// TwinCAT 3 PLC project TcForge
// Title: TcForge
// Company: Home
// ProjectVersion: 2.0.0.0
// ProgramVersion: 3.1.4026.26
// libraries:
//   Tc2_Standard, 3.4.7.0 (Beckhoff Automation GmbH)
//   Tc2_System, 3.10.2.0 (Beckhoff Automation GmbH)
//   Tc3_Module, 3.4.7.0 (Beckhoff Automation GmbH)
// project tree:
//   POUs/Control/BangBang/ ST_BangBang_Cfg.TcDUT, FB_BangBang.TcPOU
//   POUs/Control/PID/ E_ControlReason.TcDUT, ST_PID_Full_Cfg.TcDUT, ST_PID_Full_Sts.TcDUT, FB_PID_Full.TcPOU
//   POUs/Control/Temperature/ ST_TempController_Cfg.TcDUT, ST_TempController_Sts.TcDUT, FB_TempController.TcPOU
//   POUs/Control/SwitchingPV/ E_PvSource.TcDUT, ST_SwitchingPvPid_Cfg.TcDUT, ST_SwitchingPvPid_Sts.TcDUT, FB_SwitchingPvPid.TcPOU
//   POUs/Control/Hysteresis/ E_HysteresisReason.TcDUT, ST_Hysteresis_Cfg.TcDUT, ST_Hysteresis_Sts.TcDUT, FB_HysteresisControl.TcPOU
//   POUs/Utilities/ FB_ExecutionContinuity.TcPOU, F_IsFiniteReal.TcPOU, F_IsFiniteLReal.TcPOU, F_GetTaskCycleTime.TcPOU, F_Now.TcPOU (not stored), FB_BitMatrix64.TcPOU, FB_LPF_FirstOrder_IIR.TcPOU
//   POUs/IO/Common/ E_IOHealthReason.TcDUT, FB_IOQualityMonitor.TcPOU (not stored), F_EtherCATSlaveDataValid.TcPOU, E_IO_Quality.TcDUT, E_Unit.TcDUT, U_IoRaw_In.TcDUT, U_IoRaw_Out.TcDUT (not stored)
//   POUs/Base/ FB_OperatorMailbox.TcPOU, ST_OperatorCommandRecord.TcDUT (not stored), E_OperatorCommand.TcDUT, E_Requester.TcDUT (not stored), E_RpcMethodResponse.TcDUT (not stored), F_ValidateRequester.TcPOU (not stored), FB_DeviceBase.TcPOU, ST_DeviceHeader_Sts.TcDUT (not stored), ST_FaultEntry.TcDUT (not stored)
//   POUs/Devices/Pneumatics/TwoPosActuator/ E_TwoPosActuator_Fault.TcDUT (not stored), E_TwoPosActuator_State.TcDUT (not stored), FB_TwoPosActuator.TcPOU, ST_TwoPosActuator_Cfg.TcDUT (not stored), ST_TwoPosActuator_Sts.TcDUT (not stored)
//   POUs/Logic/Interlocks/ FB_Interlock.TcPOU, ST_Interlock_Config.TcDUT, ST_Interlock_Status.TcDUT, ST_Interlock_Faceplate.TcDUT
//   POUs/Logic/Sequencing/Permissives/ FB_Permissives.TcPOU, ST_Permissive_Config.TcDUT (not stored), ST_Permissive_Status.TcDUT, ST_Permissive_Faceplate.TcDUT
//   POUs/Logic/Sequencing/StateMachine/ E_SM_Fault.TcDUT, E_SM_State.TcDUT, FB_StateMachine.TcPOU, FB_Step.TcPOU, ST_SM_Status.TcDUT, ST_SM_Step.TcDUT (not stored)
//   POUs/IO/DigitalInput/ FB_DigitalInput.TcPOU, ST_DigitalInput_Cfg.TcDUT, ST_DigitalInput_Sts.TcDUT, E_DigitalInput_Fault.TcDUT (not stored)
//   POUs/IO/DigitalOutput/ FB_DigitalOutput.TcPOU, ST_DigitalOutput_Cfg.TcDUT (not stored), ST_DigitalOutput_Sts.TcDUT, E_DigitalOutput_Fault.TcDUT, E_DigitalOutput_Mode.TcDUT
//   POUs/IO/AnalogInput/ FB_AnalogInput.TcPOU, ST_AnalogInput_Cfg.TcDUT, ST_AnalogInput_Sts.TcDUT, E_AnalogInput_Fault.TcDUT (not stored)
//   POUs/IO/AnalogOutput/ FB_AnalogOutput.TcPOU, ST_AnalogOutput_Cfg.TcDUT, ST_AnalogOutput_Sts.TcDUT, E_AnalogOutput_Fault.TcDUT (not stored)
//   POUs/Alarms/Common/ I_Alarm.TcIO (not stored), E_AlarmEvaluation.TcDUT (not stored), E_AlarmSeverity.TcDUT, ST_Alarm_Cfg.TcDUT (not stored), ST_Alarm_Sts.TcDUT, FB_AlarmBase.TcPOU
//   POUs/Alarms/Simple/ ST_AlarmSimple_Cfg.TcDUT, FB_AlarmSimple.TcPOU
//   POUs/Alarms/Threshold/ ST_AlarmThreshold_Cfg.TcDUT, FB_AlarmThreshold.TcPOU
//   POUs/Alarms/Limit/ ST_AlarmLimit_Cfg.TcDUT, ST_AlarmLimit_Sts.TcDUT, FB_AlarmLimit.TcPOU
//   POUs/Alarms/Deviation/ ST_AlarmDeviation_Cfg.TcDUT, FB_AlarmDeviation.TcPOU (not stored)
//   POUs/Alarms/RateOfChange/ ST_AlarmRateOfChange_Cfg.TcDUT, FB_AlarmRateOfChange.TcPOU
// real-time tasks:
//   TASK PlcTask: cycle T#10ms, priority 1, ADS port 350

// ---- POUs/Control/BangBang/ST_BangBang_Cfg.TcDUT
// The two CV values map a Boolean demand into engineering output units.
TYPE ST_BangBang_Cfg :
STRUCT
    hysteresis : ST_Hysteresis_Cfg;
    lowValue   : REAL := 0.0;
    highValue  : REAL := 100.0;
END_STRUCT
END_TYPE

// ---- POUs/Control/PID/E_ControlReason.TcDUT
// Controller state; an output device applies the physical safe level.
{attribute 'qualified_only'}
{attribute 'strict'}
TYPE E_ControlReason :
(
    Disabled      := 0,
    Automatic     := 1,
    Manual        := 2,
    Held          := 3,
    Tracking      := 4,
    BadQuality    := 5,
    InvalidValue  := 6,
    InvalidConfig := 7,
    InvalidTiming := 8,
    ConfigChanged := 9
);
END_TYPE

// ---- POUs/Control/PID/ST_PID_Full_Cfg.TcDUT
// All rates are engineering units per second. CV and integral limits are
// output units. A zero rate disables that directional ramp.
TYPE ST_PID_Full_Cfg :
STRUCT
    kp              : REAL := 1.0;
    ki              : REAL := 0.0; // Ideal form, 1/s.
    kd              : REAL := 0.0; // Ideal form, s.
    standardForm    : BOOL := FALSE;
    integralTime    : TIME := T#0MS; // Standard form; zero disables I.
    derivativeTime  : TIME := T#0MS; // Standard form; zero disables D.
    derivativeTau   : TIME := T#0MS; // Zero disables derivative filtering.
    reverseActing   : BOOL := FALSE;

    spMin           : REAL := -1E30;
    spMax           : REAL := 1E30;
    spRateUp        : REAL := 0.0;
    spRateDown      : REAL := 0.0;

    cvMin           : REAL := 0.0;
    cvMax           : REAL := 100.0;
    cvRateUp        : REAL := 0.0;
    cvRateDown      : REAL := 0.0;
    integralMin     : REAL := -100.0;
    integralMax     : REAL := 100.0;
    safeCv          : REAL := 0.0;

    cycleTime       : TIME := T#0MS; // Zero reads the owning task period.
    maxDt           : TIME := T#1S;  // Maximum declared task interval; not a missed-cycle detector.
END_STRUCT
END_TYPE

// ---- POUs/Control/PID/ST_PID_Full_Sts.TcDUT
// Calculation diagnostics. ready is FALSE when outCv carries safeCv.
TYPE ST_PID_Full_Sts :
STRUCT
    ready        : BOOL;
    reason       : E_ControlReason := E_ControlReason.Disabled;
    saturated    : BOOL;
    spRamping    : BOOL;
    cvRamping    : BOOL;
    spRequested  : REAL;
    spApplied    : REAL;
    pv           : REAL;
    cv           : REAL;
    error        : LREAL;
    pTerm        : LREAL;
    iTerm        : LREAL;
    dTerm        : LREAL;
END_STRUCT
END_TYPE

// ---- POUs/Control/Temperature/ST_TempController_Cfg.TcDUT
// Time-proportioning output for a heater, fan or SSR. Configure pid CV as
// 0..100 percent with safeCv=0; the wrapper rejects other CV ranges.
TYPE ST_TempController_Cfg :
STRUCT
    pid                 : ST_PID_Full_Cfg;
    pwmPeriod           : TIME := T#2S;
    standbyEnabled      : BOOL := FALSE;
    standbySetpoint     : REAL := 25.0;
END_STRUCT
END_TYPE

// ---- POUs/Control/Temperature/ST_TempController_Sts.TcDUT
TYPE ST_TempController_Sts :
STRUCT
    ready          : BOOL;
    standbyActive  : BOOL;
    dutyPercent    : REAL;
    pwmOn          : BOOL;
    pid            : ST_PID_Full_Sts;
END_STRUCT
END_TYPE

// ---- POUs/Control/SwitchingPV/E_PvSource.TcDUT
{attribute 'qualified_only'}
{attribute 'strict'}
TYPE E_PvSource :
(
    PV1 := 0,
    PV2 := 1
);
END_TYPE

// ---- POUs/Control/SwitchingPV/ST_SwitchingPvPid_Cfg.TcDUT
// Each sensor can have separate tuning and SP limits. Both configurations
// must have identical CV limits and safe CV because they drive one device.
TYPE ST_SwitchingPvPid_Cfg :
STRUCT
    pv1 : ST_PID_Full_Cfg;
    pv2 : ST_PID_Full_Cfg;
END_STRUCT
END_TYPE

// ---- POUs/Control/SwitchingPV/ST_SwitchingPvPid_Sts.TcDUT
TYPE ST_SwitchingPvPid_Sts :
STRUCT
    ready             : BOOL;
    activeSource      : E_PvSource := E_PvSource.PV1;
    sourceChanged     : BOOL;
    activePv          : REAL;
    cv                : REAL;
    pid               : ST_PID_Full_Sts;
END_STRUCT
END_TYPE

// ---- POUs/Control/Hysteresis/E_HysteresisReason.TcDUT
// Why a hysteresis controller is or is not evaluating a live measurement.
{attribute 'qualified_only'}
{attribute 'strict'}
TYPE E_HysteresisReason :
(
    Disabled      := 0,
    Ready         := 1,
    BadQuality    := 2,
    InvalidValue  := 3,
    InvalidConfig := 4
);
END_TYPE

// ---- POUs/Control/Hysteresis/ST_Hysteresis_Cfg.TcDUT
// Both thresholds use the same engineering unit as the conditioned PV.
// The default equal thresholds are deliberately invalid until configured.
TYPE ST_Hysteresis_Cfg :
STRUCT
    low        : REAL := 0.0;
    high       : REAL := 0.0;
    onBelowLow : BOOL := TRUE; // TRUE for heating/fill, FALSE for cooling/vent.
END_STRUCT
END_TYPE

// ---- POUs/Control/Hysteresis/ST_Hysteresis_Sts.TcDUT
// Diagnostic status only. The application connects outDemand to an owned
// output device and remains responsible for its interlocks and safe level.
TYPE ST_Hysteresis_Sts :
STRUCT
    ready      : BOOL;
    demand     : BOOL;
    inDeadband : BOOL;
    reason     : E_HysteresisReason := E_HysteresisReason.Disabled;
END_STRUCT
END_TYPE

// ---- POUs/IO/Common/E_IOHealthReason.TcDUT
{attribute 'qualified_only'}
{attribute 'strict'}
TYPE E_IOHealthReason : (Disabled := 0, NoSample := 1, Communication := 2, Device := 3,
    InvalidSample := 4, Stale := 5, InvalidConfig := 6, SequenceReset := 7, Good := 8) USINT;
END_TYPE

// ---- POUs/Base/E_OperatorCommand.TcDUT
{attribute 'qualified_only'}
{attribute 'strict'}
TYPE E_OperatorCommand : (Reset, Ack, SetValue, ForceSafe, SetOn, SetOff, Advance, Retract, Abort, Home, Pause, Proceed, Retry, Start, Stop); END_TYPE

// ---- POUs/Logic/Interlocks/ST_Interlock_Config.TcDUT
(*
Interlock Configuration Structure
=================================
Configuration for FB_Interlock. Latching is the defining behavior of an
interlock, so every mapped bit latches by default (no nLatch mask). Bits
can optionally be made bypassable via nBypassable.
*)
{attribute 'OPC.UA.DA' := '1'}
{attribute 'OPC.UA.DA.Access' := '1'}
{attribute 'OPC.UA.DA.StructuredType' := '1'}
TYPE ST_Interlock_Config :
STRUCT
    // Required bits cannot disappear when their producer stops running.
    nRequired : ULINT := 0;
	{attribute 'OPC.UA.DA.Description' := 'Bypass configuration bitmask (1=bypassable, 0=not bypassable)'}
	nBypassable : ULINT := 0;
	{attribute 'OPC.UA.DA.Description' := 'Human readable names for each interlock bit'}
	aNames : ARRAY[0..63] OF STRING(50);
END_STRUCT
END_TYPE

// ---- POUs/Logic/Interlocks/ST_Interlock_Status.TcDUT
(*
Interlock Status Structure
==========================
Status outputs for FB_Interlock.
*)
{attribute 'OPC.UA.DA' := '1'}
{attribute 'OPC.UA.DA.Access' := '1'}
{attribute 'OPC.UA.DA.StructuredType' := '1'}
TYPE ST_Interlock_Status :
STRUCT
    nMissing : ULINT; // Required but not refreshed within the mapping timeout.
	{attribute 'OPC.UA.DA.Description' := 'Overall status - TRUE when all interlocks are good'}
	bOK : BOOL := FALSE;
	{attribute 'OPC.UA.DA.Description' := 'Effective interlock status after latch + bypass (1=good, 0=bad)'}
	nInterlocks : ULINT := 0;
	{attribute 'OPC.UA.DA.Description' := 'Latched status - stays bad until Reset() (1=good, 0=latched bad)'}
	nLatched : ULINT := 0;
	{attribute 'OPC.UA.DA.Description' := 'Current bypass mask (1=bypassed, 0=not bypassed)'}
	nBypassMask : ULINT := 0;
	{attribute 'OPC.UA.DA.Description' := 'Bit index (0-63) of the first bit to trip, 999=no trips'}
	nFirstFailureBitIndex : UDINT := 999;
	{attribute 'OPC.UA.DA.Description' := 'Individual interlock faceplate data for HMI'}
	aFaceplates : ARRAY[0..63] OF ST_Interlock_Faceplate;
END_STRUCT
END_TYPE

// ---- POUs/Logic/Interlocks/ST_Interlock_Faceplate.TcDUT
(*
Interlock Faceplate Structure
=============================
Per-bit HMI data for a single interlock condition.
*)
{attribute 'OPC.UA.DA' := '1'}
{attribute 'OPC.UA.DA.Access' := '1'}
{attribute 'OPC.UA.DA.StructuredType' := '1'}
TYPE ST_Interlock_Faceplate :
STRUCT
	{attribute 'OPC.UA.DA.Description' := 'Human readable name of the interlock'}
	name : STRING(50);
	{attribute 'OPC.UA.DA.Description' := 'Effective status after latch + bypass (TRUE=good, FALSE=bad)'}
	ok : BOOL;
	{attribute 'OPC.UA.DA.Description' := 'Raw real-time condition (TRUE=good, FALSE=bad)'}
	live : BOOL;
	{attribute 'OPC.UA.DA.Description' := 'TRUE if currently latched bad (needs Reset)'}
	latched : BOOL;
	{attribute 'OPC.UA.DA.Description' := 'TRUE if this bit is actively mapped via MapInput'}
	mapped : BOOL;
	{attribute 'OPC.UA.DA.Description' := 'TRUE if this bit is currently bypassed'}
	bypassed : BOOL;
	{attribute 'OPC.UA.DA.Description' := 'TRUE if this bit is configured as bypassable'}
	bypassable : BOOL;
END_STRUCT
END_TYPE

// ---- POUs/Logic/Sequencing/Permissives/ST_Permissive_Status.TcDUT
(*
Permissive Status Structure
===========================
Contains all status outputs from permissive function block
*)
{attribute 'OPC.UA.DA' := '1'}
{attribute 'OPC.UA.DA.Access' := '1'}
{attribute 'OPC.UA.DA.StructuredType' := '1'}
TYPE ST_Permissive_Status :
STRUCT
    nMissing : ULINT; // Required but not refreshed within the mapping timeout.
	{attribute 'OPC.UA.DA.Description' := 'Overall status - TRUE when all permissive bits are good'}
	bOK : BOOL := FALSE;
	{attribute 'OPC.UA.DA.Description' := 'Current permissive status after logic (1=good, 0=bad)'}
	nPermissives : ULINT := 0;
	{attribute 'OPC.UA.DA.Description' := 'Current bypass mask (1=bypassed, 0=not bypassed)'}
	nBypassMask : ULINT := 0;
	{attribute 'OPC.UA.DA.Description' := 'Bit index (0-63) of the first failure, 999=no failures'}
	nFirstFailureBitIndex : UDINT := 999;
	
	{attribute 'OPC.UA.DA.Description' := 'Individual permissive faceplate data for HMI'}
	aFaceplates : ARRAY[0..63] OF ST_Permissive_Faceplate;
END_STRUCT
END_TYPE

// ---- POUs/Logic/Sequencing/Permissives/ST_Permissive_Faceplate.TcDUT
(*
Permissive Faceplate Structure
==============================
Individual permissive bit information for HMI faceplate display
*)
{attribute 'OPC.UA.DA' := '1'}
{attribute 'OPC.UA.DA.Access' := '1'}
{attribute 'OPC.UA.DA.StructuredType' := '1'}
TYPE ST_Permissive_Faceplate :
STRUCT
	{attribute 'OPC.UA.DA.Description' := 'Human readable name of the permissive'}
	name : STRING(50);
	{attribute 'OPC.UA.DA.Description' := 'Real-time status of this permissive bit (TRUE=good, FALSE=bad)'}
	ok : BOOL;
	{attribute 'OPC.UA.DA.Description' := 'TRUE if this bit is actively mapped via MapInput'}
	mapped : BOOL;
	{attribute 'OPC.UA.DA.Description' := 'TRUE if this bit is currently bypassed'}
	bypassed : BOOL;
	{attribute 'OPC.UA.DA.Description' := 'TRUE if this bit is configured as bypassable'}
	bypassable : BOOL;
END_STRUCT
END_TYPE

// ---- POUs/Logic/Sequencing/StateMachine/E_SM_Fault.TcDUT
{attribute 'qualified_only'}
{attribute 'to_string'}
// Fault codes surfaced by FB_StateMachine through ST_DeviceHeader_Sts (the
// fault book-keeping lives on FB_DeviceBase). Range convention mirrors
// E_RpcMethodResponse so codes are self-documenting:
//
//   0        No fault
//   1-9      Timeouts
//   10-19    Feedback / hardware
//   20-29    State violations
//   30-39    Configuration
//   50-59    Interlocks / permissives
//   70-79    Submodule / propagation
//   100+     Device / application custom
//
// HMI displays ResolveFaultString(code) for the stable title and faultReason
// for the contextual detail (step number, step name, free-form operator
// message). Both live in ST_DeviceHeader_Sts.
TYPE E_SM_Fault :
(
    None                    := 0,

    StepTimeout             := 1,    // FB_Step.tonTimeout expired
    OddStepReached          := 2,    // default fault when a step moves onto an odd step number
    StepUserFault           := 3,    // user called step.RaiseFault(code, reason)

    InvalidStepConfiguration := 30,
    MissingStepImplementation := 31,
    DuplicateStepImplementation := 32,
    ShutdownFailed := 33,

    RunningInterlockTripped := 50,   // intlkRunning tripped, auto-aborted

    SubmoduleFaulted        := 70    // external inpSubmoduleFaulted asserted
);
END_TYPE

// ---- POUs/Logic/Sequencing/StateMachine/E_SM_State.TcDUT
{attribute 'qualified_only'}
{attribute 'strict'}
{attribute 'to_string'}
// Minimum useful set of machine states.
//
// Waiting states (quiescent, no sequence driving outputs):
//     STOPPED  - power-on default, not homed. Entry from Abort is STOPPED with Status.Faulted = TRUE.
//     READY    - homed and either just-homed or just-completed a cycle. LastState distinguishes the two.
//     PAUSED   - frozen mid-cycle, context held for Proceed.
//
// Active states (a step sequence is executing):
//     HOMING      (steps 1000-1999)
//     RUNNING     (steps 3000-3999)
//     STOPPING    (steps 2000-2999) - graceful shutdown sequence
//     ABORTING    (steps 5000-5999) - fast-safe shutdown sequence
//     PAUSING     (steps 4000-4999) - park motion / save context
//     PROCEEDING  (steps 6000-6999) - restore context / resume
TYPE E_SM_State :
(
    STOPPED     := 0,
    RUNNING     := 1,
    STOPPING    := 2,
    HOMING      := 4,
    ABORTING    := 8,
    READY       := 16,
    PAUSING     := 32,
    PAUSED      := 64,
    PROCEEDING  := 128
);
END_TYPE

// ---- POUs/Logic/Sequencing/StateMachine/ST_SM_Status.TcDUT
(*
Aggregated status published by FB_StateMachine. Contains the common device
header, the current state, derived readiness flags, OEE condition codes,
and the active step snapshot (ST_SM_Step).
*)
{attribute 'OPC.UA.DA' := '1'}
{attribute 'OPC.UA.DA.Access' := '1'}
{attribute 'OPC.UA.DA.StructuredType' := '1'}
TYPE ST_SM_Status :
STRUCT
    // Common device header (ready/busy/faulted, fault codes + strings, timestamps).
    header : ST_DeviceHeader_Sts;

    // Current state (enum with to_string for HMI)
    State : E_SM_State := E_SM_State.STOPPED;
    LastState : E_SM_State := E_SM_State.STOPPED;

    // Derived state categories
    ActiveState : BOOL;
    WaitingState : BOOL;

    // Computed fault flags
    Faulted : BOOL; // Always the base device fault state.
    AtRecoveryStep : BOOL; // Odd-numbered recovery step, independent of fault storage.
    SubmoduleFaulted : BOOL;
    ShutdownFailed : BOOL; // Abort failed; STOPPED does not imply confirmed physical shutdown.
    FailedStep : DINT; // Last failed step, cleared only by a successful Reset.

    // Permission-derived readiness
    ReadyToHome : BOOL;
    ReadyToStart : BOOL;
    ReadyToProceed : BOOL;

    // Auto-run tracking
    AutoCycleRequest : BOOL;

    // OEE condition codes (0 = clear, non-zero = active reason code)
    BlockedCondition : DINT;
    StarvedCondition : DINT;

    // Active step snapshot
    Step : ST_SM_Step;
END_STRUCT
END_TYPE

// ---- POUs/IO/DigitalInput/ST_DigitalInput_Cfg.TcDUT
// Configuration for FB_DigitalInput. All fields are configurable; defaults
// yield a plain pass-through of the physical signal.
{attribute 'OPC.UA.DA' := '1'}
{attribute 'OPC.UA.DA.Access' := '1'}
{attribute 'OPC.UA.DA.StructuredType' := '1'}
TYPE ST_DigitalInput_Cfg :
STRUCT
    // Signal conditioning
    {attribute 'OPC.UA.DA.Description' := 'Invert input signal (active-low sensors)'}
    invert            : BOOL := FALSE;

    // Asymmetric debounce: separate delays for each edge so a noisy 24 V
    // signal can have e.g. a 20 ms ON-delay but 0 ms OFF-delay. Set both to
    // T#0MS to disable.
    {attribute 'OPC.UA.DA.Description' := 'Rising-edge debounce delay (ON)'}
    debounceOn        : TIME := T#0MS;
    {attribute 'OPC.UA.DA.Description' := 'Falling-edge debounce delay (OFF)'}
    debounceOff       : TIME := T#0MS;

    // Quality watchdog: if inpQuality stays BAD for this long the FB raises
    // E_DigitalInput_Fault.BadQuality. T#0MS disables the watchdog.
    {attribute 'OPC.UA.DA.Description' := 'Raise BadQuality fault after this long in BAD quality (T#0MS = disabled)'}
    qualityFaultAfter : TIME := T#0MS;
END_STRUCT
END_TYPE

// ---- POUs/IO/DigitalInput/ST_DigitalInput_Sts.TcDUT
// Status of FB_DigitalInput. `header` is shared with every other device FB
// (see ST_DeviceHeader_Sts); device-specific fields sit below.
{attribute 'OPC.UA.DA' := '1'}
{attribute 'OPC.UA.DA.Access' := '1'}
{attribute 'OPC.UA.DA.StructuredType' := '1'}
TYPE ST_DigitalInput_Sts :
STRUCT
    header        : ST_DeviceHeader_Sts;

    {attribute 'OPC.UA.DA.Description' := 'Final processed value (after invert + debounce)'}
    value      : BOOL;
    {attribute 'OPC.UA.DA.Description' := 'Raw terminal reading (before invert / debounce)'}
    rawValue   : BOOL;
    {attribute 'OPC.UA.DA.Description' := 'Signal quality tag'}
    quality    : E_IO_Quality := E_IO_Quality.UNKNOWN;
    {attribute 'OPC.UA.DA.Description' := 'One-scan pulse on debounced rising edge'}
    risingEdge : BOOL;
    {attribute 'OPC.UA.DA.Description' := 'One-scan pulse on debounced falling edge'}
    fallingEdge: BOOL;
END_STRUCT
END_TYPE

// ---- POUs/IO/DigitalOutput/ST_DigitalOutput_Sts.TcDUT
// Status of FB_DigitalOutput. `header` is shared with every other device FB
// (see ST_DeviceHeader_Sts); device-specific fields sit below.
{attribute 'OPC.UA.DA' := '1'}
{attribute 'OPC.UA.DA.Access' := '1'}
{attribute 'OPC.UA.DA.StructuredType' := '1'}
TYPE ST_DigitalOutput_Sts :
STRUCT
    outputInhibited : BOOL;
    header        : ST_DeviceHeader_Sts;

    {attribute 'OPC.UA.DA.Description' := 'Final physical output value (after mode + invert)'}
    value      : BOOL;
    {attribute 'OPC.UA.DA.Description' := 'Last commanded value (survives power cycle)'}
    commanded  : BOOL;
    {attribute 'OPC.UA.DA.Description' := 'Signal quality tag'}
    quality    : E_IO_Quality := E_IO_Quality.UNKNOWN;
    {attribute 'OPC.UA.DA.Description' := 'One-scan pulse on physical output rising edge'}
    risingEdge : BOOL;
    {attribute 'OPC.UA.DA.Description' := 'One-scan pulse on physical output falling edge'}
    fallingEdge: BOOL;
END_STRUCT
END_TYPE

// ---- POUs/IO/AnalogInput/ST_AnalogInput_Cfg.TcDUT
// Configuration for FB_AnalogInput. Defaults provide numeric 0..100 scaling of
// an INT terminal scaled linearly from raw 0..32767 — adjust for the real
// hardware.
//
// FB_AnalogInput is intentionally conditioning-only: raw type select, quality
// gate, clamp-to-scaling-range, linear scale, optional LPF. If you need HH /
// HI / LO / LL process alarms, compose FB_AlarmLimit with the published
// value — that keeps alarm config, latching, severity, and ack logic in
// one place (see docs/8-Alarms.md).
{attribute 'OPC.UA.DA' := '1'}
{attribute 'OPC.UA.DA.Access' := '1'}
{attribute 'OPC.UA.DA.StructuredType' := '1'}
TYPE ST_AnalogInput_Cfg :
STRUCT
    // Which UNION member to read. Supported values:
    //   TYPE_REAL, TYPE_INT, TYPE_UINT, TYPE_WORD, TYPE_DWORD, TYPE_UDINT, TYPE_DINT
    {attribute 'OPC.UA.DA.Description' := 'Terminal numeric type (selects UNION member)'}
    inputType          : __SYSTEM.TYPE_CLASS := __SYSTEM.TYPE_CLASS.TYPE_INT;

    // When TRUE, the FB skips clamping + scaling + filtering and publishes
    // the raw REAL representation directly. Handy for soft signals, bit-
    // masked terminals, or diagnostics.
    {attribute 'OPC.UA.DA.Description' := 'Bypass clamp + scale + filter; publish raw value'}
    useRawValue        : BOOL := FALSE;

    // Raw-to-EU linear scaling. Example: 4-20 mA on an EL3024 reports raw
    // in [0, 32767]; to get 0-100 % set fRawMin=0, fRawMax=32767, fPvMin=0,
    // fPvMax=100.
    {attribute 'OPC.UA.DA.Description' := 'Raw value corresponding to fPvMin'}
    rawMin             : REAL := 0.0;
    {attribute 'OPC.UA.DA.Description' := 'Raw value corresponding to fPvMax'}
    rawMax             : REAL := 32767.0;

    {attribute 'OPC.UA.DA.Description' := 'Engineering value at fRawMin'}
    euMin              : REAL := 0.0;
    {attribute 'OPC.UA.DA.Description' := 'Engineering value at fRawMax'}
    euMax              : REAL := 100.0;
    {attribute 'OPC.UA.DA.Description' := 'Engineering-unit display metadata; configure explicitly'}
    unit               : E_Unit := E_Unit.UNSPECIFIED;

    // Clamp reporting. sts.clamped* always tracks whether the raw input
    // was outside [rawMin, rawMax]; clampAsFault promotes that condition
    // to a persistent device fault.
    {attribute 'OPC.UA.DA.Description' := 'Promote out-of-range raw readings to ClampLow / ClampHigh faults'}
    clampAsFault       : BOOL := FALSE;

    // Optional first-order low-pass filter. T#0MS disables filtering.
    {attribute 'OPC.UA.DA.Description' := 'Low-pass filter time constant (T#0MS = disabled)'}
    filterTau          : TIME := T#0MS;

    // Quality watchdog.
    {attribute 'OPC.UA.DA.Description' := 'Raise BadQuality fault after this long in BAD quality (T#0MS = disabled)'}
    qualityFaultAfter  : TIME := T#0MS;
END_STRUCT
END_TYPE

// ---- POUs/IO/AnalogInput/ST_AnalogInput_Sts.TcDUT
// Status of FB_AnalogInput. `header` is shared with every device FB;
// device-specific fields sit below. Process-alarm status (HH/HI/LO/LL) is
// not part of this surface — use FB_AlarmLimit composed with value.
{attribute 'OPC.UA.DA' := '1'}
{attribute 'OPC.UA.DA.Access' := '1'}
{attribute 'OPC.UA.DA.StructuredType' := '1'}
TYPE ST_AnalogInput_Sts :
STRUCT
    header          : ST_DeviceHeader_Sts;

    {attribute 'OPC.UA.DA.Description' := 'Final value in engineering units (after clamp, scale, filter)'}
    value        : REAL;
    {attribute 'OPC.UA.DA.Description' := 'Raw value as REAL, before clamping and scaling'}
    rawReal      : REAL;
    {attribute 'OPC.UA.DA.Description' := 'Scaled value (EU), before filter'}
    scaled       : REAL;
    {attribute 'OPC.UA.DA.Description' := 'Echo of cfg.unit for HMI consumption'}
    unit         : E_Unit := E_Unit.UNSPECIFIED;
    {attribute 'OPC.UA.DA.Description' := 'Signal quality tag (may be promoted to CLAMPED)'}
    quality      : E_IO_Quality := E_IO_Quality.UNKNOWN;

    {attribute 'OPC.UA.DA.Description' := 'Raw below configured RawMin'}
    clampedLow   : BOOL;
    {attribute 'OPC.UA.DA.Description' := 'Raw above configured RawMax'}
    clampedHigh  : BOOL;
    {attribute 'OPC.UA.DA.Description' := 'Either clamp direction active'}
    clampActive  : BOOL;
END_STRUCT
END_TYPE

// ---- POUs/IO/AnalogOutput/ST_AnalogOutput_Cfg.TcDUT
// Configuration for FB_AnalogOutput. Defaults drive a numeric 0..100 command
// range into an INT 0..32767 scaled terminal.
{attribute 'OPC.UA.DA' := '1'}
{attribute 'OPC.UA.DA.Access' := '1'}
{attribute 'OPC.UA.DA.StructuredType' := '1'}
TYPE ST_AnalogOutput_Cfg :
STRUCT
    // Startup restoration requires explicit application opt-in.
    restoreCommandOnRestart : BOOL := FALSE;
    // Optional hold during bad/unknown quality. Recovery still requires a fresh command.
    holdOnBadQuality : BOOL := FALSE;
    safeRaw : REAL := 0.0; // Terminal units, independent of scaling.
    // Which UNION member to write. Supported values:
    //   TYPE_REAL, TYPE_INT, TYPE_UINT, TYPE_WORD, TYPE_DWORD, TYPE_UDINT, TYPE_DINT
    {attribute 'OPC.UA.DA.Description' := 'Terminal numeric type (selects UNION member)'}
    outputType         : __SYSTEM.TYPE_CLASS := __SYSTEM.TYPE_CLASS.TYPE_INT;

    // When TRUE, the FB writes the command REAL directly into the UNION
    // without clamping or scaling. Handy for soft signals / diagnostics.
    {attribute 'OPC.UA.DA.Description' := 'Write commanded value directly; skip clamp + scale'}
    useRawValue        : BOOL := FALSE;

    // Command limits in engineering units.
    {attribute 'OPC.UA.DA.Description' := 'Minimum allowed command (EU)'}
    minCv              : REAL := 0.0;
    {attribute 'OPC.UA.DA.Description' := 'Maximum allowed command (EU)'}
    maxCv              : REAL := 100.0;

    // EU <-> raw linear scaling.
    {attribute 'OPC.UA.DA.Description' := 'Engineering value at fRawMin'}
    euMin              : REAL := 0.0;
    {attribute 'OPC.UA.DA.Description' := 'Engineering value at fRawMax'}
    euMax              : REAL := 100.0;
    {attribute 'OPC.UA.DA.Description' := 'Raw value at fEuMin'}
    rawMin             : REAL := 0.0;
    {attribute 'OPC.UA.DA.Description' := 'Raw value at fEuMax'}
    rawMax             : REAL := 32767.0;
    {attribute 'OPC.UA.DA.Description' := 'Engineering-unit display metadata; configure explicitly'}
    unit               : E_Unit := E_Unit.UNSPECIFIED;

    // Clamp alarm behaviour.
    {attribute 'OPC.UA.DA.Description' := 'Promote clamping to a device fault (ClampLow / ClampHigh)'}
    clampAsFault       : BOOL := FALSE;

    // Quality watchdog.
    {attribute 'OPC.UA.DA.Description' := 'Raise BadQuality fault after this long in BAD quality (T#0MS = disabled)'}
    qualityFaultAfter  : TIME := T#0MS;
END_STRUCT
END_TYPE

// ---- POUs/IO/AnalogOutput/ST_AnalogOutput_Sts.TcDUT
// Status of FB_AnalogOutput. `header` is shared with every device FB;
// device-specific fields sit below.
{attribute 'OPC.UA.DA' := '1'}
{attribute 'OPC.UA.DA.Access' := '1'}
{attribute 'OPC.UA.DA.StructuredType' := '1'}
TYPE ST_AnalogOutput_Sts :
STRUCT
    outputInhibited : BOOL; // value (EU) is not valid when inhibited; rawReal is the applied fallback/held raw value.
    header        : ST_DeviceHeader_Sts;

    {attribute 'OPC.UA.DA.Description' := 'Clamped command actually written (EU)'}
    value      : REAL;
    {attribute 'OPC.UA.DA.Description' := 'Last commanded value before clamping (EU, survives power cycle)'}
    commanded  : REAL;
    {attribute 'OPC.UA.DA.Description' := 'Raw value written to the terminal (REAL view of the UNION)'}
    rawReal    : REAL;
    {attribute 'OPC.UA.DA.Description' := 'Echo of cfg.unit for HMI consumption'}
    unit       : E_Unit := E_Unit.UNSPECIFIED;
    {attribute 'OPC.UA.DA.Description' := 'Signal quality tag'}
    quality    : E_IO_Quality := E_IO_Quality.UNKNOWN;

    {attribute 'OPC.UA.DA.Description' := 'Command clamped at MinCv'}
    clampedLow : BOOL;
    {attribute 'OPC.UA.DA.Description' := 'Command clamped at MaxCv'}
    clampedHigh: BOOL;
    {attribute 'OPC.UA.DA.Description' := 'Either clamp direction active'}
    clampActive: BOOL;
END_STRUCT
END_TYPE

// ---- POUs/IO/DigitalOutput/E_DigitalOutput_Fault.TcDUT
{attribute 'qualified_only'}
{attribute 'to_string'}
// Fault codes for FB_DigitalOutput. Range convention matches the shared
// device-fault convention (see docs/2-Architecture.md):
//   0        No fault
//   1-9      Timeouts
//   10-19    Feedback / hardware / signal
//   20-29    State violations
//   40-49    Configuration / process limits
//   50-59    Interlocks / permissives
TYPE E_DigitalOutput_Fault :
(
    None        := 0,

    BadConfig := 40,
    BadQuality  := 10     // outgoing signal not writable (quality latched BAD past cfg.tQualityFaultAfter)
);
END_TYPE

// ---- POUs/IO/DigitalOutput/E_DigitalOutput_Mode.TcDUT
// Output shaping modes for FB_DigitalOutput.
//   Regular         : output tracks the commanded value (optionally inverted)
//   SinglePulse     : one-shot — commanded rising edge drives the output ON
//                     for cfg.tPulseOn, then OFF
//   ContinuousPulse : while commanded TRUE, output cycles ON/OFF with
//                     cfg.tPulseOn / cfg.tPulseOff (good for lamps, blinkers,
//                     repeat-start pulses)
{attribute 'qualified_only'}
{attribute 'strict'}
{attribute 'to_string'}
TYPE E_DigitalOutput_Mode :
(
    Regular         := 0,
    SinglePulse     := 1,
    ContinuousPulse := 2
);
END_TYPE

// ---- POUs/IO/Common/E_IO_Quality.TcDUT
// Signal quality tag carried by every IO block's status. The value lets the
// HMI and downstream logic react to wire breaks, out-of-range readings, or
// sensor faults without each consumer reinventing its own "is this bit /
// reading trustworthy?" logic.
//
// Meaning:
//   UNKNOWN : block has not evaluated yet (first scan, or no data source)
//   BAD     : signal is not usable (wire break, TwinCAT WcState, etc.)
//   GOOD    : signal is valid and within configured range
//   CLAMPED : signal is valid but was forced to the scaling limit
//
// Some device inputs default to GOOD for software signals. Hardware applications
// must explicitly supply quality from diagnostics, e.g. FB_IOQualityMonitor.
{attribute 'qualified_only'}
{attribute 'strict'}
{attribute 'to_string'}
TYPE E_IO_Quality :
(
    UNKNOWN := 0,
    BAD     := 1,
    GOOD    := 2,
    CLAMPED := 3
) USINT;
END_TYPE

// ---- POUs/IO/Common/E_Unit.TcDUT
// Display metadata for analog IO. The value is already scaled by the owning
// device; this enum does not convert or validate engineering units. An HMI may
// map the enum to a symbol (for example MILLIMETER -> mm).
//
// Keep explicit numeric values stable after publication because OPC clients may
// store them. Extend for machine-relevant measurements; never repurpose a code.
{attribute 'qualified_only'}
{attribute 'strict'}
{attribute 'to_string'}
TYPE E_Unit :
(
    // A channel whose display unit has not been configured.
    UNSPECIFIED                   := 0,

    // Ratio and discrete quantity.
    PERCENT                       := 1,     // %
    COUNT                         := 2,     // pieces / cycles

    // Position, orientation, velocity and acceleration.
    MILLIMETER                    := 3,     // mm
    MICROMETER                    := 4,     // um
    DEGREE                        := 5,     // angular degrees
    MILLIMETER_PER_SECOND         := 6,     // mm/s
    MILLIMETER_PER_SECOND_SQUARED := 7,     // mm/s^2
    RPM                           := 8,     // revolutions/minute

    // Force, torque, mass and pneumatic pressure.
    NEWTON                        := 9,     // N
    NEWTON_METER                  := 10,    // N m
    GRAM                          := 11,    // g
    KILOGRAM                      := 12,    // kg
    BAR                           := 13,    // bar
    KILOPASCAL                    := 14,    // kPa

    // Temperature and electrical measurements.
    DEGREE_CELSIUS                := 15,    // deg C
    DEGREE_FAHRENHEIT             := 16,    // deg F
    VOLTS                         := 17,    // V
    AMPS                          := 18,    // A
    WATT                          := 19,    // W
    HERTZ                         := 20,    // Hz

    // Cycle measurements and sensor-reported durations.
    SECOND                        := 21,    // s
    MILLISECOND                   := 22     // ms
);
END_TYPE

// ---- POUs/IO/Common/U_IoRaw_In.TcDUT
// Raw terminal representation. The application owns hardware mapping.
TYPE U_IoRaw_In :
UNION
    dw    : DWORD;
    fReal : REAL;
    w     : WORD;
    nInt  : INT;
    ui    : UINT;
    di    : DINT;
    udi   : UDINT;
END_UNION
END_TYPE

// ---- POUs/Alarms/Common/E_AlarmSeverity.TcDUT
// HMI / stacklight severity tag carried by every alarm status.
// Numeric order is meaningful — aggregators MAX() across alarms to pick the
// highest tier that's currently active.
{attribute 'qualified_only'}
{attribute 'strict'}
{attribute 'to_string'}
TYPE E_AlarmSeverity :
(
    NONE     := 0,   // bookkeeping: alarm disabled or inactive
    INFO     := 1,   // informational, no operator action required
    WARNING  := 2,   // operator should investigate
    CRITICAL := 3,   // urgent; process may be about to lose control
    SHUTDOWN := 4    // interlock-grade; a controller is already acting
) USINT;
END_TYPE

// ---- POUs/Alarms/Common/ST_Alarm_Sts.TcDUT
// Uniform alarm status. Every FB_Alarm* fills this struct identically so
// HMIs and aggregators can bind to any alarm generically.
{attribute 'OPC.UA.DA' := '1'}
{attribute 'OPC.UA.DA.Access' := '1'}
{attribute 'OPC.UA.DA.StructuredType' := '1'}
TYPE ST_Alarm_Sts :
STRUCT
    // Valid fresh evaluation; active may remain held while validity is false.
    valid : BOOL;
    evaluationState : E_AlarmEvaluation := E_AlarmEvaluation.Disabled;
    {attribute 'OPC.UA.DA.Description' := 'Echo of cfg.bEnable'}
    enabled    : BOOL;

    {attribute 'OPC.UA.DA.Description' := 'Instantaneous condition before debounce'}
    raw        : BOOL;

    {attribute 'OPC.UA.DA.Description' := 'After tOnDelay / tOffDelay'}
    debounced  : BOOL;

    {attribute 'OPC.UA.DA.Description' := 'Public is-it-firing bit (latch when bRequireAck)'}
    active     : BOOL;

    {attribute 'OPC.UA.DA.Description' := 'TRUE while latch is awaiting Ack()'}
    latched    : BOOL;

    {attribute 'OPC.UA.DA.Description' := 'TRUE once the current latch has been acknowledged'}
    acked      : BOOL;

    {attribute 'OPC.UA.DA.Description' := 'Severity while active; NONE while inactive'}
    eSeverity     : E_AlarmSeverity := E_AlarmSeverity.NONE;

    {attribute 'OPC.UA.DA.Description' := 'Echo of cfg.sMessage'}
    sMessage      : STRING(79);

    {attribute 'OPC.UA.DA.Description' := 'Who acknowledged the current latch'}
    ackRequester  : E_Requester;

    {attribute 'OPC.UA.DA.Description' := 'Last rising edge of debounced (LTIME)'}
    tsTripped     : LTIME;

    {attribute 'OPC.UA.DA.Description' := 'Last falling edge of debounced (LTIME)'}
    tsCleared     : LTIME;

    {attribute 'OPC.UA.DA.Description' := 'Last accepted Ack() timestamp (LTIME)'}
    tsAcked       : LTIME;
END_STRUCT
END_TYPE

// ---- POUs/Alarms/Simple/ST_AlarmSimple_Cfg.TcDUT
// Config for FB_AlarmSimple — no extra knobs beyond the shared common head.
{attribute 'OPC.UA.DA' := '1'}
{attribute 'OPC.UA.DA.Access' := '1'}
{attribute 'OPC.UA.DA.StructuredType' := '1'}
TYPE ST_AlarmSimple_Cfg :
STRUCT
    {attribute 'OPC.UA.DA.Description' := 'Shared alarm configuration (enable, delays, ack, severity, message)'}
    common : ST_Alarm_Cfg;
END_STRUCT
END_TYPE

// ---- POUs/Alarms/Threshold/ST_AlarmThreshold_Cfg.TcDUT
// Config for FB_AlarmThreshold. Single-direction REAL threshold check.
// Rule: strict > / < (exact threshold value does not trip).
// Exactly one direction must be selected while enabled; otherwise InvalidConfig.
{attribute 'OPC.UA.DA' := '1'}
{attribute 'OPC.UA.DA.Access' := '1'}
{attribute 'OPC.UA.DA.StructuredType' := '1'}
TYPE ST_AlarmThreshold_Cfg :
STRUCT
    {attribute 'OPC.UA.DA.Description' := 'Shared alarm configuration'}
    common     : ST_Alarm_Cfg;

    {attribute 'OPC.UA.DA.Description' := 'Threshold value to compare inpValue against'}
    fThreshold : REAL := 0.0;

    {attribute 'OPC.UA.DA.Description' := 'TRUE = trip when inpValue > fThreshold'}
    bFailHigh  : BOOL := FALSE;

    {attribute 'OPC.UA.DA.Description' := 'TRUE = trip when inpValue < fThreshold'}
    bFailLow   : BOOL := FALSE;
END_STRUCT
END_TYPE

// ---- POUs/Alarms/Limit/ST_AlarmLimit_Cfg.TcDUT
// Four-level limit ladder: HiHi / Hi / Lo / LoLo. Each level is a full
// ST_AlarmThreshold_Cfg, so each can have its own delay, severity, ack
// requirement, and message. Remember every level defaults to bEnable := FALSE.
{attribute 'OPC.UA.DA' := '1'}
{attribute 'OPC.UA.DA.Access' := '1'}
{attribute 'OPC.UA.DA.StructuredType' := '1'}
TYPE ST_AlarmLimit_Cfg :
STRUCT
    {attribute 'OPC.UA.DA.Description' := 'High-High (critical high, e.g. emergency shutdown)'}
    HiHi : ST_AlarmThreshold_Cfg;

    {attribute 'OPC.UA.DA.Description' := 'High (warning high, operator alert)'}
    Hi   : ST_AlarmThreshold_Cfg;

    {attribute 'OPC.UA.DA.Description' := 'Low (warning low)'}
    Lo   : ST_AlarmThreshold_Cfg;

    {attribute 'OPC.UA.DA.Description' := 'Low-Low (critical low)'}
    LoLo : ST_AlarmThreshold_Cfg;
END_STRUCT
END_TYPE

// ---- POUs/Alarms/Limit/ST_AlarmLimit_Sts.TcDUT
// Status for FB_AlarmLimit. Each level has its own raw ST_Alarm_Sts so the
// HMI can show full forensics per tier. The top-level *Suppressed* flags apply
// flooding suppression: HiHi suppresses Hi, LoLo suppresses Lo — so the HMI
// can pick exactly one active level per direction.
{attribute 'OPC.UA.DA' := '1'}
{attribute 'OPC.UA.DA.Access' := '1'}
{attribute 'OPC.UA.DA.StructuredType' := '1'}
TYPE ST_AlarmLimit_Sts :
STRUCT
    // Valid fresh evaluation; active may remain held while validity is false.
    valid : BOOL;
    evaluationState : E_AlarmEvaluation := E_AlarmEvaluation.Disabled;
    {attribute 'OPC.UA.DA.Description' := 'HiHi sub-alarm status'}
    HiHi : ST_Alarm_Sts;
    {attribute 'OPC.UA.DA.Description' := 'Hi sub-alarm status'}
    Hi   : ST_Alarm_Sts;
    {attribute 'OPC.UA.DA.Description' := 'Lo sub-alarm status'}
    Lo   : ST_Alarm_Sts;
    {attribute 'OPC.UA.DA.Description' := 'LoLo sub-alarm status'}
    LoLo : ST_Alarm_Sts;

    {attribute 'OPC.UA.DA.Description' := 'HiHi active (rollup after suppression)'}
    hiHiActive : BOOL;
    {attribute 'OPC.UA.DA.Description' := 'Hi active and not suppressed by HiHi'}
    hiActive   : BOOL;
    {attribute 'OPC.UA.DA.Description' := 'Lo active and not suppressed by LoLo'}
    loActive   : BOOL;
    {attribute 'OPC.UA.DA.Description' := 'LoLo active (rollup after suppression)'}
    loLoActive : BOOL;

    {attribute 'OPC.UA.DA.Description' := 'Any of the four levels currently active'}
    anyActive  : BOOL;
    {attribute 'OPC.UA.DA.Description' := 'Highest severity across all active levels'}
    eSeverity     : E_AlarmSeverity;
END_STRUCT
END_TYPE

// ---- POUs/Alarms/Deviation/ST_AlarmDeviation_Cfg.TcDUT
// Config for FB_AlarmDeviation. Two modes, selected by bUseSetpoint.
//
//   Absolute (bUseSetpoint = FALSE, default):
//       trip = inpPv > fHighLimit OR inpPv < fLowLimit
//       inpSetpoint is ignored
//
//   Setpoint deviation (bUseSetpoint = TRUE):
//       trip = inpPv > (inpSetpoint + fHighLimit) OR inpPv < (inpSetpoint - fLowLimit)
//       High/Low limits are asymmetric deviations from setpoint.
{attribute 'OPC.UA.DA' := '1'}
{attribute 'OPC.UA.DA.Access' := '1'}
{attribute 'OPC.UA.DA.StructuredType' := '1'}
TYPE ST_AlarmDeviation_Cfg :
STRUCT
    {attribute 'OPC.UA.DA.Description' := 'Shared alarm configuration'}
    common       : ST_Alarm_Cfg;

    {attribute 'OPC.UA.DA.Description' := 'Absolute high limit, or +deviation when bUseSetpoint = TRUE'}
    fHighLimit   : REAL := 0.0;

    {attribute 'OPC.UA.DA.Description' := 'Absolute low limit, or -deviation when bUseSetpoint = TRUE'}
    fLowLimit    : REAL := 0.0;

    {attribute 'OPC.UA.DA.Description' := 'TRUE = limits are relative to inpSetpoint'}
    bUseSetpoint : BOOL := FALSE;
END_STRUCT
END_TYPE

// ---- POUs/Alarms/RateOfChange/ST_AlarmRateOfChange_Cfg.TcDUT
// Config for FB_AlarmRateOfChange. Rate limit in engineering-units per second.
// The check is symmetric — ABS(rate) > fRateLimit — so it catches runaway
// both ways (sensor drop, control saturation, exothermic runaway…).
{attribute 'OPC.UA.DA' := '1'}
{attribute 'OPC.UA.DA.Access' := '1'}
{attribute 'OPC.UA.DA.StructuredType' := '1'}
TYPE ST_AlarmRateOfChange_Cfg :
STRUCT
    {attribute 'OPC.UA.DA.Description' := 'Shared alarm configuration'}
    common     : ST_Alarm_Cfg;

    {attribute 'OPC.UA.DA.Description' := 'Max allowable |rate of change| in units per second'}
    fRateLimit : REAL := 0.0;
END_STRUCT
END_TYPE

// ---- POUs/Control/BangBang/FB_BangBang.TcPOU
// Numeric bang-bang control composed from the quality-gated hysteresis core.
// The application/output device owns manual commands, hold and safe terminal
// level; no retained request, source handler or RPC can bypass the cyclic owner.
FUNCTION_BLOCK FB_BangBang
VAR_INPUT
    enable      : BOOL;
    pv          : REAL;
    pvQuality   : E_IO_Quality := E_IO_Quality.UNKNOWN;
    cfg         : ST_BangBang_Cfg;
END_VAR
VAR_OUTPUT
    outCv       : REAL;
    outDemand   : BOOL;
    sts         : ST_Hysteresis_Sts;
END_VAR
VAR
    _hysteresis : FB_HysteresisControl;
END_VAR

// A bad numeric mapping must clear the internal hysteresis state too.
IF NOT F_IsFiniteReal(value := cfg.lowValue)
    OR NOT F_IsFiniteReal(value := cfg.highValue) THEN
    _hysteresis(enable := FALSE);
    outCv := 0.0;
    outDemand := FALSE;
    sts := _hysteresis.sts;
    sts.reason := E_HysteresisReason.InvalidConfig;
    RETURN;
END_IF;

_hysteresis(
    enable := enable,
    pv := pv,
    pvQuality := pvQuality,
    cfg := cfg.hysteresis
);
sts := _hysteresis.sts;
outDemand := _hysteresis.outDemand;

IF NOT sts.ready THEN
    outCv := 0.0;
ELSIF outDemand THEN
    outCv := cfg.highValue;
ELSE
    outCv := cfg.lowValue;
END_IF;

END_FUNCTION_BLOCK

// ---- POUs/Control/Hysteresis/FB_HysteresisControl.TcPOU
// Quality-gated two-threshold demand for an owned discrete output.
// Call once from the same cyclic task as the PV conditioner and output device.
// Loss of enable, usable PV, or configuration de-energizes demand; recovery
// never inherits the previous ON state while the PV is inside the deadband.
// This block does not switch physical IO or implement operator RPCs.
FUNCTION_BLOCK FB_HysteresisControl
VAR_INPUT
    enable    : BOOL;
    pv        : REAL;
    pvQuality : E_IO_Quality := E_IO_Quality.UNKNOWN;
    cfg       : ST_Hysteresis_Cfg;
END_VAR
VAR_OUTPUT
    outDemand : BOOL;
    sts       : ST_Hysteresis_Sts;
END_VAR
VAR
    _haveConfig : BOOL;
    _lastCfg    : ST_Hysteresis_Cfg;
END_VAR

// Any unusable input takes the same OFF path. Validate floating-point bits
// before comparisons: a signaling NaN can fault a TwinCAT task when compared.
sts.ready := FALSE;
sts.inDeadband := FALSE;

IF NOT enable THEN
    outDemand := FALSE;
    _haveConfig := FALSE;
    sts.reason := E_HysteresisReason.Disabled;
ELSIF NOT F_IsFiniteReal(value := cfg.low)
    OR NOT F_IsFiniteReal(value := cfg.high) THEN
    outDemand := FALSE;
    _haveConfig := FALSE;
    sts.reason := E_HysteresisReason.InvalidConfig;
ELSIF cfg.low >= cfg.high THEN
    outDemand := FALSE;
    _haveConfig := FALSE;
    sts.reason := E_HysteresisReason.InvalidConfig;
ELSIF pvQuality <> E_IO_Quality.GOOD THEN
    outDemand := FALSE;
    _haveConfig := FALSE;
    sts.reason := E_HysteresisReason.BadQuality;
ELSIF NOT F_IsFiniteReal(value := pv) THEN
    outDemand := FALSE;
    _haveConfig := FALSE;
    sts.reason := E_HysteresisReason.InvalidValue;
ELSE
    // A changed threshold or direction starts from OFF. At either boundary
    // the fresh PV then determines the new demand; within the band it stays OFF.
    IF NOT _haveConfig
        OR cfg.low <> _lastCfg.low
        OR cfg.high <> _lastCfg.high
        OR cfg.onBelowLow <> _lastCfg.onBelowLow THEN
        outDemand := FALSE;
        _lastCfg := cfg;
        _haveConfig := TRUE;
    END_IF;

    IF cfg.onBelowLow THEN
        IF pv <= cfg.low THEN
            outDemand := TRUE;
        ELSIF pv >= cfg.high THEN
            outDemand := FALSE;
        END_IF;
    ELSE
        IF pv >= cfg.high THEN
            outDemand := TRUE;
        ELSIF pv <= cfg.low THEN
            outDemand := FALSE;
        END_IF;
    END_IF;

    sts.ready := TRUE;
    sts.inDeadband := pv > cfg.low AND pv < cfg.high;
    sts.reason := E_HysteresisReason.Ready;
END_IF;

sts.demand := outDemand;

END_FUNCTION_BLOCK

// ---- POUs/Utilities/F_IsFiniteReal.TcPOU
// IEEE-754 classification by integer exponent bits; no floating-point operation.
// Safe with runtime floating-point exceptions enabled, including signaling NaNs.
FUNCTION F_IsFiniteReal : BOOL
VAR_INPUT value : REAL; END_VAR
VAR bits : DWORD; END_VAR

Tc2_System.MEMCPY(destAddr := ADR(bits), srcAddr := ADR(value), n := SIZEOF(bits));
F_IsFiniteReal := (bits AND DWORD#16#7F800000) <> DWORD#16#7F800000;

END_FUNCTION

// ---- POUs/Control/PID/FB_PID_Full.TcPOU
// Cyclic PID calculation; the application owns setpoint/mode requests, source
// arbitration, IO mapping and interlocks. No RPC or persistent output intent.
// Invalid quality/configuration/timing returns the configured safe CV and
// discards integral/derivative history. Call once per owning task cycle.
FUNCTION_BLOCK FB_PID_Full
VAR_INPUT
    enable      : BOOL;
    pv          : REAL;
    pvQuality   : E_IO_Quality := E_IO_Quality.UNKNOWN;
    setpoint    : REAL;
    manual      : BOOL;
    manualCv    : REAL;
    hold        : BOOL;
    track       : BOOL; // One-scan transfer from another controller.
    trackCv     : REAL;
    cfg         : ST_PID_Full_Cfg;
END_VAR
VAR_OUTPUT
    outCv       : REAL;
    sts         : ST_PID_Full_Sts;
END_VAR
VAR
    _initialized : BOOL;
    _lastCfg     : ST_PID_Full_Cfg;
    _sp          : LREAL;
    _cv          : LREAL;
    _integral    : LREAL;
    _derivative  : LREAL;
    _prevPv      : LREAL;

    cycleDuration : TIME;
    dtSec        : LREAL;
    spTarget     : LREAL;
    delta        : LREAL;
    gainI        : LREAL;
    gainD        : LREAL;
    direction    : LREAL;
    error        : LREAL;
    pTerm        : LREAL;
    dRaw         : LREAL;
    candidateI   : LREAL;
    unsaturated  : LREAL;
    targetCv     : LREAL;
END_VAR

// Initialize the published status before each possible early return.
sts.ready := FALSE;
sts.reason := E_ControlReason.Disabled;
sts.saturated := FALSE;
sts.spRamping := FALSE;
sts.cvRamping := FALSE;
sts.spRequested := 0.0;
sts.spApplied := 0.0;
sts.pv := 0.0;
sts.error := 0.0;
sts.pTerm := 0.0;
sts.iTerm := 0.0;
sts.dTerm := 0.0;
outCv := 0.0;

// Bit-classify every REAL before any numeric comparison or arithmetic.
IF NOT ValidConfig() THEN
    ResetState();
    sts.reason := E_ControlReason.InvalidConfig;
    sts.cv := outCv;
    RETURN;
END_IF;

outCv := cfg.safeCv;
IF NOT enable THEN
    ResetState();
    sts.cv := outCv;
    RETURN;
END_IF;

IF pvQuality <> E_IO_Quality.GOOD THEN
    ResetState();
    sts.reason := E_ControlReason.BadQuality;
    sts.cv := outCv;
    RETURN;
END_IF;

IF NOT F_IsFiniteReal(value := pv)
    OR NOT F_IsFiniteReal(value := setpoint)
    OR (manual AND NOT F_IsFiniteReal(value := manualCv))
    OR (track AND NOT F_IsFiniteReal(value := trackCv)) THEN
    ResetState();
    sts.reason := E_ControlReason.InvalidValue;
    sts.cv := outCv;
    RETURN;
END_IF;

cycleDuration := cfg.cycleTime;
IF cycleDuration = T#0MS THEN
    cycleDuration := F_GetTaskCycleTime();
END_IF;
IF cycleDuration = T#0MS OR cycleDuration > cfg.maxDt THEN
    ResetState();
    sts.reason := E_ControlReason.InvalidTiming;
    sts.cv := outCv;
    RETURN;
END_IF;
dtSec := TIME_TO_REAL(cycleDuration) / 1000.0;

// Tuning or limit edits remove the old controller history for one scan.
IF _initialized AND ChangedConfig() THEN
    ResetState();
    sts.reason := E_ControlReason.ConfigChanged;
    sts.cv := outCv;
    RETURN;
END_IF;

spTarget := setpoint;
IF spTarget < cfg.spMin THEN spTarget := cfg.spMin; END_IF;
IF spTarget > cfg.spMax THEN spTarget := cfg.spMax; END_IF;

IF NOT _initialized THEN
    _sp := spTarget;
    _cv := cfg.safeCv;
    _integral := 0.0;
    _derivative := 0.0;
    _prevPv := pv;
    _lastCfg := cfg;
    _initialized := TRUE;
END_IF;

// Limit setpoint motion in physical engineering units per second.
delta := spTarget - _sp;
IF delta > 0.0 AND cfg.spRateUp > 0.0 THEN
    IF delta > cfg.spRateUp * dtSec THEN delta := cfg.spRateUp * dtSec; END_IF;
ELSIF delta < 0.0 AND cfg.spRateDown > 0.0 THEN
    IF -delta > cfg.spRateDown * dtSec THEN delta := -cfg.spRateDown * dtSec; END_IF;
END_IF;
_sp := _sp + delta;

direction := 1.0;
IF cfg.reverseActing THEN direction := -1.0; END_IF;
error := direction * (_sp - pv);
pTerm := cfg.kp * error;

gainI := cfg.ki;
gainD := cfg.kd;
IF cfg.standardForm THEN
    gainI := 0.0;
    IF cfg.integralTime > T#0MS THEN
        gainI := cfg.kp / (TIME_TO_REAL(cfg.integralTime) / 1000.0);
    END_IF;
    gainD := cfg.kp * (TIME_TO_REAL(cfg.derivativeTime) / 1000.0);
END_IF;

// Derivative on measurement prevents a setpoint step from kicking the CV.
dRaw := -direction * gainD * ((pv - _prevPv) / dtSec);
_prevPv := pv;
IF cfg.derivativeTau > T#0MS THEN
    delta := dtSec / ((TIME_TO_REAL(cfg.derivativeTau) / 1000.0) + dtSec);
    _derivative := (1.0 - delta) * _derivative + delta * dRaw;
ELSE
    _derivative := dRaw;
END_IF;

// Tracking is a one-cycle bumpless handoff. Manual mode updates the integral
// bias so a later return to automatic begins at the manual CV.
IF track OR manual THEN
    IF track THEN targetCv := trackCv; ELSE targetCv := manualCv; END_IF;
    IF targetCv < cfg.cvMin THEN targetCv := cfg.cvMin; END_IF;
    IF targetCv > cfg.cvMax THEN targetCv := cfg.cvMax; END_IF;
    _cv := targetCv;
    _integral := targetCv - pTerm - _derivative;
    IF _integral < cfg.integralMin THEN _integral := cfg.integralMin; END_IF;
    IF _integral > cfg.integralMax THEN _integral := cfg.integralMax; END_IF;
    IF track THEN sts.reason := E_ControlReason.Tracking;
    ELSE sts.reason := E_ControlReason.Manual; END_IF;
ELSIF hold THEN
    sts.reason := E_ControlReason.Held;
ELSE
    // Integrate only as far as the CV boundary. Rejecting the whole step can
    // strand the CV just below its limit due to floating-point rounding.
    candidateI := _integral + gainI * error * dtSec;
    IF candidateI < cfg.integralMin THEN candidateI := cfg.integralMin; END_IF;
    IF candidateI > cfg.integralMax THEN candidateI := cfg.integralMax; END_IF;
    unsaturated := pTerm + candidateI + _derivative;
    sts.saturated := unsaturated > cfg.cvMax OR unsaturated < cfg.cvMin;
    IF unsaturated > cfg.cvMax AND candidateI > _integral THEN
        candidateI := cfg.cvMax - pTerm - _derivative;
        IF candidateI < _integral THEN candidateI := _integral; END_IF;
    ELSIF unsaturated < cfg.cvMin AND candidateI < _integral THEN
        candidateI := cfg.cvMin - pTerm - _derivative;
        IF candidateI > _integral THEN candidateI := _integral; END_IF;
    END_IF;
    _integral := candidateI;

    unsaturated := pTerm + _integral + _derivative;
    targetCv := unsaturated;
    IF targetCv < cfg.cvMin THEN targetCv := cfg.cvMin; END_IF;
    IF targetCv > cfg.cvMax THEN targetCv := cfg.cvMax; END_IF;
    sts.saturated := sts.saturated OR targetCv <> unsaturated;

    delta := targetCv - _cv;
    IF delta > 0.0 AND cfg.cvRateUp > 0.0 THEN
        IF delta > cfg.cvRateUp * dtSec THEN delta := cfg.cvRateUp * dtSec; END_IF;
    ELSIF delta < 0.0 AND cfg.cvRateDown > 0.0 THEN
        IF -delta > cfg.cvRateDown * dtSec THEN delta := -cfg.cvRateDown * dtSec; END_IF;
    END_IF;
    _cv := _cv + delta;
    sts.cvRamping := _cv <> targetCv;
    sts.reason := E_ControlReason.Automatic;
END_IF;

// All published REAL values are inside validated REAL limits.
outCv := LREAL_TO_REAL(_cv);
sts.ready := TRUE;
sts.spRamping := _sp <> spTarget;
sts.spRequested := setpoint;
sts.spApplied := LREAL_TO_REAL(_sp);
sts.pv := pv;
sts.cv := outCv;
sts.error := error;
sts.pTerm := pTerm;
sts.iTerm := _integral;
sts.dTerm := _derivative;

METHOD PRIVATE ResetState
_initialized := FALSE;
_sp := 0.0;
_cv := outCv;
_integral := 0.0;
_derivative := 0.0;
_prevPv := 0.0;
END_METHOD

METHOD PRIVATE ValidConfig : BOOL
ValidConfig := F_IsFiniteReal(value := cfg.kp)
    AND F_IsFiniteReal(value := cfg.ki)
    AND F_IsFiniteReal(value := cfg.kd)
    AND F_IsFiniteReal(value := cfg.spMin)
    AND F_IsFiniteReal(value := cfg.spMax)
    AND F_IsFiniteReal(value := cfg.spRateUp)
    AND F_IsFiniteReal(value := cfg.spRateDown)
    AND F_IsFiniteReal(value := cfg.cvMin)
    AND F_IsFiniteReal(value := cfg.cvMax)
    AND F_IsFiniteReal(value := cfg.cvRateUp)
    AND F_IsFiniteReal(value := cfg.cvRateDown)
    AND F_IsFiniteReal(value := cfg.integralMin)
    AND F_IsFiniteReal(value := cfg.integralMax)
    AND F_IsFiniteReal(value := cfg.safeCv);
IF NOT ValidConfig THEN RETURN; END_IF;

ValidConfig := cfg.kp >= 0.0 AND cfg.ki >= 0.0 AND cfg.kd >= 0.0
    AND cfg.spMin < cfg.spMax
    AND cfg.cvMin < cfg.cvMax
    AND cfg.integralMin < cfg.integralMax
    AND cfg.spRateUp >= 0.0 AND cfg.spRateDown >= 0.0
    AND cfg.cvRateUp >= 0.0 AND cfg.cvRateDown >= 0.0
    AND cfg.safeCv >= cfg.cvMin AND cfg.safeCv <= cfg.cvMax
    AND cfg.maxDt > T#0MS;
END_METHOD

METHOD PRIVATE ChangedConfig : BOOL
ChangedConfig := cfg.kp <> _lastCfg.kp
    OR cfg.ki <> _lastCfg.ki OR cfg.kd <> _lastCfg.kd
    OR cfg.standardForm <> _lastCfg.standardForm
    OR cfg.integralTime <> _lastCfg.integralTime
    OR cfg.derivativeTime <> _lastCfg.derivativeTime
    OR cfg.derivativeTau <> _lastCfg.derivativeTau
    OR cfg.reverseActing <> _lastCfg.reverseActing
    OR cfg.spMin <> _lastCfg.spMin OR cfg.spMax <> _lastCfg.spMax
    OR cfg.spRateUp <> _lastCfg.spRateUp OR cfg.spRateDown <> _lastCfg.spRateDown
    OR cfg.cvMin <> _lastCfg.cvMin OR cfg.cvMax <> _lastCfg.cvMax
    OR cfg.cvRateUp <> _lastCfg.cvRateUp OR cfg.cvRateDown <> _lastCfg.cvRateDown
    OR cfg.integralMin <> _lastCfg.integralMin
    OR cfg.integralMax <> _lastCfg.integralMax
    OR cfg.safeCv <> _lastCfg.safeCv
    OR cfg.cycleTime <> _lastCfg.cycleTime
    OR cfg.maxDt <> _lastCfg.maxDt;
END_METHOD

END_FUNCTION_BLOCK

// ---- POUs/Utilities/F_GetTaskCycleTime.TcPOU
// Returns the cycle time of the calling task as a TIME value (ms resolution).
// Useful for filters and ramps that need `dt` in physical units rather than
// PLC scans.
//
// Internally: TwinCAT stores CycleTime as UDINT in units of 100 ns, so we
// divide by 10_000 to convert to ms before casting to TIME.
FUNCTION F_GetTaskCycleTime : TIME
// Per-call storage: different owning tasks must not share a cached task index.
VAR
    fbGetCurTaskIndex : GETCURTASKINDEX;
END_VAR

fbGetCurTaskIndex();
F_GetTaskCycleTime := UDINT_TO_TIME(
    TwinCAT_SystemInfoVarList._TaskInfo[fbGetCurTaskIndex.index].CycleTime / 10_000
);

END_FUNCTION

// ---- POUs/Control/Temperature/FB_TempController.TcPOU
// Composes full PID with a bounded time-proportioning output. No physical
// terminal is written here. The application must route outOn through a safe
// owned output device and qualify its independent overtemperature protection.
FUNCTION_BLOCK FB_TempController
VAR_INPUT
    enable       : BOOL;
    pv           : REAL;
    pvQuality    : E_IO_Quality := E_IO_Quality.UNKNOWN;
    setpoint     : REAL;
    standby      : BOOL;
    manual       : BOOL;
    manualDuty   : REAL;
    hold         : BOOL;
    cfg          : ST_TempController_Cfg;
END_VAR
VAR_OUTPUT
    outDuty      : REAL;
    outOn        : BOOL;
    sts          : ST_TempController_Sts;
END_VAR
VAR
    _pid         : FB_PID_Full;
    _phaseMs     : LREAL;
    _lastPeriod  : TIME;
    _periodKnown : BOOL;
    selectedSp   : REAL;
    cycleDuration : TIME;
    periodMs     : LREAL;
END_VAR

sts.ready := FALSE;
sts.standbyActive := cfg.standbyEnabled AND standby;
sts.dutyPercent := 0.0;
sts.pwmOn := FALSE;
outDuty := 0.0;
outOn := FALSE;

// Validate the output interpretation before passing any command to PID.
IF NOT F_IsFiniteReal(value := cfg.standbySetpoint)
    OR NOT F_IsFiniteReal(value := cfg.pid.cvMin)
    OR NOT F_IsFiniteReal(value := cfg.pid.cvMax)
    OR NOT F_IsFiniteReal(value := cfg.pid.safeCv) THEN
    _pid(enable := FALSE);
    _phaseMs := 0.0;
    sts.pid := _pid.sts;
    RETURN;
END_IF;

IF cfg.pid.cvMin <> 0.0 OR cfg.pid.cvMax <> 100.0
    OR cfg.pid.safeCv <> 0.0
    OR cfg.pwmPeriod < T#100MS OR cfg.pwmPeriod > T#1H THEN
    _pid(enable := FALSE);
    _phaseMs := 0.0;
    sts.pid := _pid.sts;
    RETURN;
END_IF;

selectedSp := setpoint;
IF sts.standbyActive THEN selectedSp := cfg.standbySetpoint; END_IF;

_pid(
    enable := enable,
    pv := pv,
    pvQuality := pvQuality,
    setpoint := selectedSp,
    manual := manual,
    manualCv := manualDuty,
    hold := hold,
    track := FALSE,
    cfg := cfg.pid
);
sts.pid := _pid.sts;

IF NOT _pid.sts.ready THEN
    _phaseMs := 0.0;
    _periodKnown := FALSE;
    RETURN;
END_IF;

cycleDuration := cfg.pid.cycleTime;
IF cycleDuration = T#0MS THEN cycleDuration := F_GetTaskCycleTime(); END_IF;
IF cycleDuration = T#0MS OR cycleDuration > cfg.pid.maxDt THEN
    _phaseMs := 0.0;
    RETURN;
END_IF;

IF NOT _periodKnown OR cfg.pwmPeriod <> _lastPeriod THEN
    _phaseMs := 0.0;
    _lastPeriod := cfg.pwmPeriod;
    _periodKnown := TRUE;
ELSE
    _phaseMs := _phaseMs + TIME_TO_REAL(cycleDuration);
END_IF;

periodMs := TIME_TO_REAL(cfg.pwmPeriod);
WHILE _phaseMs >= periodMs DO
    _phaseMs := _phaseMs - periodMs;
END_WHILE;

outDuty := _pid.outCv;
outOn := outDuty > 0.0 AND _phaseMs < (outDuty / 100.0) * periodMs;
sts.ready := TRUE;
sts.dutyPercent := outDuty;
sts.pwmOn := outOn;

END_FUNCTION_BLOCK

// ---- POUs/Control/SwitchingPV/FB_SwitchingPvPid.TcPOU
// Selects one of two independently tuned PID channels for one owned CV.
// Inactive history is cleared every scan. A source change tracks the last
// valid CV for one scan, then the selected controller resumes regulation.
// Source authority belongs to the application, not this calculation block.
FUNCTION_BLOCK FB_SwitchingPvPid
VAR_INPUT
    enable      : BOOL;
    source      : E_PvSource := E_PvSource.PV1;
    pv1         : REAL;
    quality1    : E_IO_Quality := E_IO_Quality.UNKNOWN;
    setpoint1   : REAL;
    pv2         : REAL;
    quality2    : E_IO_Quality := E_IO_Quality.UNKNOWN;
    setpoint2   : REAL;
    manual      : BOOL;
    manualCv    : REAL;
    hold        : BOOL;
    cfg         : ST_SwitchingPvPid_Cfg;
END_VAR
VAR_OUTPUT
    outCv       : REAL;
    sts         : ST_SwitchingPvPid_Sts;
END_VAR
VAR
    _pid1          : FB_PID_Full;
    _pid2          : FB_PID_Full;
    _haveSelection : BOOL;
    _lastSource    : E_PvSource := E_PvSource.PV1;
    _lastCv        : REAL;
    changed        : BOOL;
END_VAR

sts.ready := FALSE;
sts.sourceChanged := FALSE;
sts.activeSource := source;
sts.activePv := 0.0;
sts.cv := 0.0;
outCv := 0.0;

// A single output device cannot reinterpret its safe value or CV range when
// the selected measurement changes. Reject mismatched output contracts.
IF NOT F_IsFiniteReal(value := cfg.pv1.cvMin)
    OR NOT F_IsFiniteReal(value := cfg.pv1.cvMax)
    OR NOT F_IsFiniteReal(value := cfg.pv1.safeCv)
    OR NOT F_IsFiniteReal(value := cfg.pv2.cvMin)
    OR NOT F_IsFiniteReal(value := cfg.pv2.cvMax)
    OR NOT F_IsFiniteReal(value := cfg.pv2.safeCv) THEN
    _pid1(enable := FALSE);
    _pid2(enable := FALSE);
    _haveSelection := FALSE;
    RETURN;
END_IF;

IF cfg.pv1.cvMin <> cfg.pv2.cvMin
    OR cfg.pv1.cvMax <> cfg.pv2.cvMax
    OR cfg.pv1.safeCv <> cfg.pv2.safeCv THEN
    _pid1(enable := FALSE);
    _pid2(enable := FALSE);
    _haveSelection := FALSE;
    RETURN;
END_IF;

IF NOT enable THEN
    _pid1(enable := FALSE);
    _pid2(enable := FALSE);
    _haveSelection := FALSE;
    _lastCv := cfg.pv1.safeCv;
    outCv := _lastCv;
    sts.cv := outCv;
    RETURN;
END_IF;

changed := _haveSelection AND source <> _lastSource;
sts.sourceChanged := changed;

IF source = E_PvSource.PV1 THEN
    _pid2(enable := FALSE);
    _pid1(
        enable := TRUE,
        pv := pv1,
        pvQuality := quality1,
        setpoint := setpoint1,
        manual := manual,
        manualCv := manualCv,
        hold := hold,
        track := changed,
        trackCv := _lastCv,
        cfg := cfg.pv1
    );
    outCv := _pid1.outCv;
    sts.pid := _pid1.sts;
    sts.activePv := pv1;
ELSIF source = E_PvSource.PV2 THEN
    _pid1(enable := FALSE);
    _pid2(
        enable := TRUE,
        pv := pv2,
        pvQuality := quality2,
        setpoint := setpoint2,
        manual := manual,
        manualCv := manualCv,
        hold := hold,
        track := changed,
        trackCv := _lastCv,
        cfg := cfg.pv2
    );
    outCv := _pid2.outCv;
    sts.pid := _pid2.sts;
    sts.activePv := pv2;
ELSE
    _pid1(enable := FALSE);
    _pid2(enable := FALSE);
    _haveSelection := FALSE;
    RETURN;
END_IF;

sts.ready := sts.pid.ready;
sts.cv := outCv;
_lastCv := outCv;
_lastSource := source;
_haveSelection := sts.ready;

END_FUNCTION_BLOCK

// ---- POUs/Utilities/FB_ExecutionContinuity.TcPOU
// Application supplies the owning system task identity/counter and PLC online-change counter.
// A pulse requires application cancellation and explicit recovery; no output is controlled here.
FUNCTION_BLOCK FB_ExecutionContinuity
VAR_INPUT
    taskIndex : DINT;
    cycleCounter, onlineChangeCounter : UDINT;
    // Application policy; FALSE permits a compatible online edit, never a real gap.
    recoverOnOnlineChange : BOOL := TRUE;
END_VAR
VAR_OUTPUT interrupted, executionInterrupted, onlineChanged : BOOL; END_VAR
VAR known : BOOL; lastTask : DINT; lastCycle, lastChange, expectedCycle : UDINT; END_VAR

interrupted := FALSE;
executionInterrupted := FALSE; onlineChanged := FALSE;
IF taskIndex <= 0 THEN interrupted := TRUE; executionInterrupted := TRUE; known := FALSE; RETURN; END_IF;
IF known THEN
    IF lastCycle = UDINT#16#FFFFFFFF THEN expectedCycle := 0; ELSE expectedCycle := lastCycle + 1; END_IF;
    onlineChanged := onlineChangeCounter <> lastChange;
    executionInterrupted := taskIndex <> lastTask OR
        (cycleCounter <> lastCycle AND cycleCounter <> expectedCycle);
END_IF;
interrupted := executionInterrupted OR (onlineChanged AND recoverOnOnlineChange);
lastTask := taskIndex; lastCycle := cycleCounter; lastChange := onlineChangeCounter; known := TRUE;

END_FUNCTION_BLOCK

// ---- POUs/Utilities/F_IsFiniteLReal.TcPOU
// IEEE-754 classification by integer exponent bits; no floating-point operation.
// Safe with runtime floating-point exceptions enabled, including signaling NaNs.
FUNCTION F_IsFiniteLReal : BOOL
VAR_INPUT value : LREAL; END_VAR
VAR bits : LWORD; END_VAR

Tc2_System.MEMCPY(destAddr := ADR(bits), srcAddr := ADR(value), n := SIZEOF(bits));
F_IsFiniteLReal := (bits AND LWORD#16#7FF0000000000000) <> LWORD#16#7FF0000000000000;

END_FUNCTION

// ---- POUs/IO/Common/F_EtherCATSlaveDataValid.TcPOU
// Original mapping of documented Beckhoff InfoData.State and WcState.
// See docs/15-IO-Diagnostics.md. Link the actual slave diagnostic symbols in the application.
FUNCTION F_EtherCATSlaveDataValid : BOOL
VAR_INPUT
    diagnosticsAvailable : BOOL;
    wcState : BOOL := TRUE;
    slaveState : WORD;
END_VAR

// Low nibble: OP. Error/identity/missing/link flags invalidate data.
// Upper nibble reports communication ports, not error severity.
F_EtherCATSlaveDataValid := diagnosticsAvailable AND NOT wcState
    AND ((slaveState AND WORD#16#000F) = WORD#16#0008)
    AND ((slaveState AND WORD#16#0F30) = WORD#16#0000);

END_FUNCTION

// ---- POUs/Base/FB_OperatorMailbox.TcPOU
// One pending command, eight bounded result records. All RPC access uses TestAndSet.
// The caller supplies a nonzero request ID unique across clients and PLC restarts.
// This volatile mailbox is not a durable delivery or exactly-once service.
FUNCTION_BLOCK FB_OperatorMailbox
VAR_OUTPUT
    ownerTask : DINT;
    lastExecutionTask : DINT;
    ownershipConflict : BOOL;
END_VAR
VAR
    _lock : BOOL;
    _records : ARRAY[1..8] OF ST_OperatorCommandRecord;
    _next : UINT := 1;
    _pending : UINT;
    _executing : UINT;
    _cancelNormal : BOOL;
    _cancelSetOff : BOOL;
END_VAR

// Infrastructure methods only; the device body owns consumption.

METHOD PRIVATE Priority : UINT
VAR_INPUT command : E_OperatorCommand; END_VAR
CASE command OF
E_OperatorCommand.Abort, E_OperatorCommand.ForceSafe: Priority := 4;
E_OperatorCommand.Stop, E_OperatorCommand.SetOff: Priority := 3;
E_OperatorCommand.Reset: Priority := 2;
E_OperatorCommand.Ack, E_OperatorCommand.SetValue, E_OperatorCommand.SetOn,
E_OperatorCommand.Advance, E_OperatorCommand.Retract, E_OperatorCommand.Home,
E_OperatorCommand.Pause, E_OperatorCommand.Proceed, E_OperatorCommand.Retry,
E_OperatorCommand.Start: Priority := 1;
ELSE Priority := 0;
END_CASE;
END_METHOD

METHOD PUBLIC Submit : E_RpcMethodResponse
VAR_INPUT requestId : ULINT; command : E_OperatorCommand; value : REAL; END_VAR
VAR i : UINT; priorityValue : UINT; END_VAR
Submit := E_RpcMethodResponse.REJECTED_INVALID_PARAMETER;
priorityValue := Priority(command);
IF requestId = 0 OR priorityValue = 0 THEN RETURN; END_IF;
IF command = E_OperatorCommand.SetValue THEN
    IF NOT F_IsFiniteReal(value) THEN RETURN; END_IF;
END_IF;
Submit := E_RpcMethodResponse.REJECTED_BUSY;
IF NOT Tc2_System.TestAndSet(_lock) THEN RETURN; END_IF;
IF ownershipConflict THEN
    Submit := E_RpcMethodResponse.REJECTED_WRONG_TASK;
ELSIF ownerTask = 0 THEN
    Submit := E_RpcMethodResponse.REJECTED_NOT_READY;
ELSE
    FOR i := 1 TO 8 DO
        IF _records[i].requestId = requestId THEN
            Submit := E_RpcMethodResponse.REJECTED_DUPLICATE_REQUEST;
            _lock := FALSE; RETURN;
        END_IF;
    END_FOR;
    IF NOT ((_cancelNormal AND priorityValue < 3) OR (_cancelSetOff AND command = E_OperatorCommand.SetOff)) THEN
        IF _pending = 0 OR_ELSE priorityValue > Priority(_records[_pending].command) THEN
            IF _pending <> 0 THEN _records[_pending].result := E_RpcMethodResponse.CANCELLED; END_IF;
            _records[_next].requestId := requestId;
            _records[_next].command := command;
            _records[_next].value := value;
            _records[_next].result := E_RpcMethodResponse.QUEUED;
            _pending := _next;
            _next := _next MOD 8 + 1;
            Submit := E_RpcMethodResponse.QUEUED;
        END_IF;
    END_IF;
END_IF;
_lock := FALSE;
END_METHOD

METHOD PUBLIC GetResult : E_RpcMethodResponse
VAR_INPUT requestId : ULINT; END_VAR
VAR i : UINT; END_VAR
GetResult := E_RpcMethodResponse.REJECTED_INVALID_PARAMETER;
IF requestId = 0 THEN RETURN; END_IF;
GetResult := E_RpcMethodResponse.REJECTED_BUSY;
IF NOT Tc2_System.TestAndSet(_lock) THEN RETURN; END_IF;
GetResult := E_RpcMethodResponse.REJECTED_UNKNOWN_REQUEST;
FOR i := 1 TO 8 DO
    IF _records[i].requestId = requestId THEN GetResult := _records[i].result; EXIT; END_IF;
END_FOR;
_lock := FALSE;
END_METHOD

METHOD PUBLIC CancelNormal
VAR_INPUT
    // SetOff can energize an inverted output; configuration invalidation cancels it too.
    includeSetOff : BOOL := FALSE;
END_VAR
// Owning-task-only barrier. BOOL store is atomic; BeginConsume reconciles under the lock.
// A concurrent submission either sees this barrier or is cancelled before consumption.
_cancelNormal := TRUE;
IF includeSetOff THEN _cancelSetOff := TRUE; END_IF;
END_METHOD

METHOD PUBLIC BeginConsume : BOOL
VAR_OUTPUT command : E_OperatorCommand; value : REAL; END_VAR
VAR current : DINT; END_VAR
BeginConsume := FALSE;
current := Tc2_System.GETCURTASKINDEXEX();
IF current <= 0 THEN RETURN; END_IF;
IF NOT Tc2_System.TestAndSet(_lock) THEN RETURN; END_IF;
IF ownerTask = 0 THEN ownerTask := current; END_IF;
IF current <> ownerTask THEN ownershipConflict := TRUE; END_IF;
IF ownershipConflict THEN
    IF _pending <> 0 THEN _records[_pending].result := E_RpcMethodResponse.CANCELLED; _pending := 0; END_IF;
    _lock := FALSE; RETURN;
END_IF;
IF _cancelNormal OR _cancelSetOff THEN
    IF _pending <> 0 THEN
        IF (_cancelNormal AND Priority(_records[_pending].command) < 3) OR
           (_cancelSetOff AND _records[_pending].command = E_OperatorCommand.SetOff) THEN
            _records[_pending].result := E_RpcMethodResponse.CANCELLED; _pending := 0;
        END_IF;
    END_IF;
    _cancelNormal := FALSE;
    _cancelSetOff := FALSE;
END_IF;
IF _pending = 0 THEN _lock := FALSE; RETURN; END_IF;
_executing := _pending; _pending := 0;
command := _records[_executing].command; value := _records[_executing].value;
BeginConsume := TRUE;
// Keep the lock through the bounded owner dispatch. RPC callers return BUSY; none wait.
// Caller MUST pair every TRUE result with EndConsume, including rejected commands.
END_METHOD

METHOD PUBLIC EndConsume
VAR_INPUT result : E_RpcMethodResponse; END_VAR
IF _executing = 0 THEN RETURN; END_IF;
_records[_executing].result := result;
lastExecutionTask := Tc2_System.GETCURTASKINDEXEX();
_executing := 0;
_lock := FALSE;
END_METHOD

END_FUNCTION_BLOCK

// ---- POUs/Devices/Pneumatics/TwoPosActuator/FB_TwoPosActuator.TcPOU
{attribute 'OPC.UA.DA' := '1'}
FUNCTION_BLOCK FB_TwoPosActuator EXTENDS FB_DeviceBase
VAR_INPUT
    {attribute 'OPC.UA.DA' := '0'}
    inAdvanced : BOOL;
    {attribute 'OPC.UA.DA' := '0'}
    inRetracted : BOOL;
    {attribute 'OPC.UA.DA' := '1'}
    {attribute 'OPC.UA.DA.Access' := '1'}
    cfg : ST_TwoPosActuator_Cfg;
    cfgAdvancePermissives : ST_Permissive_Config;
    cfgRetractPermissives : ST_Permissive_Config;
END_VAR

VAR_OUTPUT
    {attribute 'OPC.UA.DA' := '1'}
    {attribute 'OPC.UA.DA.Access' := '1'}
    outAdvance : BOOL;
    {attribute 'OPC.UA.DA' := '1'}
    {attribute 'OPC.UA.DA.Access' := '1'}
    outRetract : BOOL;
    {attribute 'OPC.UA.DA' := '1'}
    {attribute 'OPC.UA.DA.Access' := '1'}
    sts : ST_TwoPosActuator_Sts;
END_VAR

VAR
    _configurationKnown : BOOL;
    _lastConfiguration : ST_TwoPosActuator_Cfg;
    _inhibited : BOOL := TRUE;
    _abortPending : BOOL;
    _advancedFeedback : BOOL;
    _retractedFeedback : BOOL;

    // Composed permissive handlers (visible on OPC under the FB instance).
    advancePermissives : FB_Permissives;
    retractPermissives : FB_Permissives;

    // Internal state tracking
    {attribute 'OPC.UA.DA' := '0'}
    currentState : E_TwoPosActuator_State := E_TwoPosActuator_State.Undefined;
    {attribute 'OPC.UA.DA' := '0'}
    previousState : E_TwoPosActuator_State;

    // Motion timers
    {attribute 'OPC.UA.DA' := '0'}
    advanceTimer : TON;
    {attribute 'OPC.UA.DA' := '0'}
    retractTimer : TON;

    // Edge detection for one-shot outputs
    {attribute 'OPC.UA.DA' := '0'}
    rTrigAdvanced : R_TRIG;
    {attribute 'OPC.UA.DA' := '0'}
    rTrigRetracted : R_TRIG;

    {attribute 'OPC.UA.DA' := '0'}
    bothFeedbackActive : BOOL;
END_VAR

_SyncConfiguration();
_ProcessOperatorCommands();
//-----------------------------------------------------------------------------
// Cyclic monitoring. Commands are issued via methods; this body only watches
// for completion/faults and keeps sts in sync. Fault latching + last-fault
// history live in FB_DeviceBase (_Raise / _ClearFault).
//-----------------------------------------------------------------------------
_advancedFeedback := inAdvanced;
_retractedFeedback := inRetracted;
advancePermissives(cfg := cfgAdvancePermissives);
retractPermissives(cfg := cfgRetractPermissives);

bothFeedbackActive := _advancedFeedback AND _retractedFeedback;

previousState := currentState;
IF (currentState = E_TwoPosActuator_State.Advancing AND NOT advancePermissives.sts.bOK) OR
   (currentState = E_TwoPosActuator_State.Retracting AND NOT retractPermissives.sts.bOK) THEN
    _Raise(code := E_TwoPosActuator_Fault.PermissivesNotOK, source := 'PERMISSIVES', reason := 'Travel condition missing or false');
    currentState := E_TwoPosActuator_State.Fault;
END_IF;

CASE currentState OF

    E_TwoPosActuator_State.Undefined:
        outAdvance := FALSE;
        outRetract := FALSE;

        IF bothFeedbackActive THEN
            currentState := E_TwoPosActuator_State.Fault;
            _Raise(
                code   := E_TwoPosActuator_Fault.BothFeedbackOn,
                source := 'FEEDBACK',
                reason := 'Both advanced and retracted feedback asserted simultaneously'
            );
        ELSIF _advancedFeedback AND NOT _retractedFeedback THEN
            currentState := E_TwoPosActuator_State.Advanced;
        ELSIF _retractedFeedback AND NOT _advancedFeedback THEN
            currentState := E_TwoPosActuator_State.Retracted;
        END_IF;

    E_TwoPosActuator_State.Retracted:
        IF cfg.holdAtRetracted THEN
            outRetract := TRUE;
        ELSE
            outRetract := FALSE;
        END_IF;
        outAdvance := FALSE;

        IF bothFeedbackActive THEN
            currentState := E_TwoPosActuator_State.Fault;
            _Raise(
                code   := E_TwoPosActuator_Fault.BothFeedbackOn,
                source := 'FEEDBACK',
                reason := 'Both advanced and retracted feedback asserted simultaneously'
            );
        ELSIF NOT _retractedFeedback THEN
            currentState := E_TwoPosActuator_State.Fault;
            _Raise(
                code   := E_TwoPosActuator_Fault.UndefinedState,
                source := 'FEEDBACK',
                reason := 'Retracted feedback lost after reaching position'
            );
        END_IF;

    E_TwoPosActuator_State.Advancing:
        outAdvance := TRUE;
        outRetract := FALSE;
        advanceTimer(IN := TRUE, PT := DINT_TO_TIME(INT_TO_DINT(cfg.advTimeoutS) * 1000));

        IF _advancedFeedback AND NOT _retractedFeedback THEN
            currentState := E_TwoPosActuator_State.Advanced;
            advanceTimer(IN := FALSE);
        ELSIF advanceTimer.Q THEN
            currentState := E_TwoPosActuator_State.Fault;
            _Raise(
                code   := E_TwoPosActuator_Fault.AdvanceTimeout,
                source := 'MOTION',
                reason := 'inFbkAdvanced did not assert within advTimeoutS'
            );
            advanceTimer(IN := FALSE);
        ELSIF bothFeedbackActive THEN
            currentState := E_TwoPosActuator_State.Fault;
            _Raise(
                code   := E_TwoPosActuator_Fault.BothFeedbackOn,
                source := 'FEEDBACK',
                reason := 'Both advanced and retracted feedback asserted while advancing'
            );
            advanceTimer(IN := FALSE);
        ELSIF NOT advancePermissives.sts.bOK THEN
            currentState := E_TwoPosActuator_State.Fault;
            _Raise(
                code   := E_TwoPosActuator_Fault.PermissivesNotOK,
                source := 'PERMISSIVES',
                reason := 'Advance permissive dropped during travel'
            );
            advanceTimer(IN := FALSE);
        END_IF;

    E_TwoPosActuator_State.Advanced:
        IF cfg.holdAtAdvanced THEN
            outAdvance := TRUE;
        ELSE
            outAdvance := FALSE;
        END_IF;
        outRetract := FALSE;

        IF bothFeedbackActive THEN
            currentState := E_TwoPosActuator_State.Fault;
            _Raise(
                code   := E_TwoPosActuator_Fault.BothFeedbackOn,
                source := 'FEEDBACK',
                reason := 'Both advanced and retracted feedback asserted simultaneously'
            );
        ELSIF NOT _advancedFeedback THEN
            currentState := E_TwoPosActuator_State.Fault;
            _Raise(
                code   := E_TwoPosActuator_Fault.UndefinedState,
                source := 'FEEDBACK',
                reason := 'Advanced feedback lost after reaching position'
            );
        END_IF;

    E_TwoPosActuator_State.Retracting:
        outRetract := TRUE;
        outAdvance := FALSE;
        retractTimer(IN := TRUE, PT := DINT_TO_TIME(INT_TO_DINT(cfg.retTimeoutS) * 1000));

        IF _retractedFeedback AND NOT _advancedFeedback THEN
            currentState := E_TwoPosActuator_State.Retracted;
            retractTimer(IN := FALSE);
        ELSIF retractTimer.Q THEN
            currentState := E_TwoPosActuator_State.Fault;
            _Raise(
                code   := E_TwoPosActuator_Fault.RetractTimeout,
                source := 'MOTION',
                reason := 'inFbkRetracted did not assert within retTimeoutS'
            );
            retractTimer(IN := FALSE);
        ELSIF bothFeedbackActive THEN
            currentState := E_TwoPosActuator_State.Fault;
            _Raise(
                code   := E_TwoPosActuator_Fault.BothFeedbackOn,
                source := 'FEEDBACK',
                reason := 'Both advanced and retracted feedback asserted while retracting'
            );
            retractTimer(IN := FALSE);
        ELSIF NOT retractPermissives.sts.bOK THEN
            currentState := E_TwoPosActuator_State.Fault;
            _Raise(
                code   := E_TwoPosActuator_Fault.PermissivesNotOK,
                source := 'PERMISSIVES',
                reason := 'Retract permissive dropped during travel'
            );
            retractTimer(IN := FALSE);
        END_IF;

    E_TwoPosActuator_State.Fault:
        outAdvance := FALSE;
        outRetract := FALSE;
        advanceTimer(IN := FALSE);
        retractTimer(IN := FALSE);
END_CASE;

IF cfg.advTimeoutS <= 0 OR cfg.retTimeoutS <= 0 THEN
    _Raise(code := E_TwoPosActuator_Fault.BadConfig, source := 'CONFIG', reason := 'Travel timeouts must be positive');
    currentState := E_TwoPosActuator_State.Fault;
END_IF;
IF NOT _inhibited AND ((currentState = E_TwoPosActuator_State.Advanced AND cfg.holdAtAdvanced AND NOT advancePermissives.sts.bOK) OR
   (currentState = E_TwoPosActuator_State.Retracted AND cfg.holdAtRetracted AND NOT retractPermissives.sts.bOK)) THEN
    _Raise(code := E_TwoPosActuator_Fault.PermissivesNotOK, source := 'PERMISSIVES', reason := 'Hold permissive missing');
    currentState := E_TwoPosActuator_State.Fault;
END_IF;
// Apply outputs from the FINAL state so a trip removes coils in the detecting scan.
IF IsFaulted() OR _inhibited OR currentState = E_TwoPosActuator_State.Undefined THEN
    outAdvance := FALSE; outRetract := FALSE;
ELSE
    outAdvance := currentState = E_TwoPosActuator_State.Advancing OR (currentState = E_TwoPosActuator_State.Advanced AND cfg.holdAtAdvanced);
    outRetract := currentState = E_TwoPosActuator_State.Retracting OR (currentState = E_TwoPosActuator_State.Retracted AND cfg.holdAtRetracted);
END_IF;

//-------------------------------------------------------------------------
// Device-specific status
// Abort priority lasts through application of the next scan.
_abortPending := FALSE;
//-------------------------------------------------------------------------
sts.state        := currentState;
sts.advanced  := (currentState = E_TwoPosActuator_State.Advanced);
sts.retracted := (currentState = E_TwoPosActuator_State.Retracted);
sts.moving    := (currentState = E_TwoPosActuator_State.Advancing) OR
                    (currentState = E_TwoPosActuator_State.Retracting);

rTrigAdvanced(CLK := sts.advanced);
sts.osAdvanced := rTrigAdvanced.Q;

rTrigRetracted(CLK := sts.retracted);
sts.osRetracted := rTrigRetracted.Q;

//-------------------------------------------------------------------------
// Common header — delegated to the base; fault/source/timestamps filled from
// the inherited fault book-keeping and source lock. busy mirrors sts.moving.
//-------------------------------------------------------------------------
_UpdateHeader(
    header      := sts.header,
    stateString := _StateToString(state := currentState),
    busy     := sts.moving
);

METHOD PUBLIC Advance : E_RpcMethodResponse
VAR_INPUT
    eRequester : E_Requester := E_Requester.PROG;
END_VAR
// Reject invalid identity before any command-specific mutation.
Advance := F_ValidateRequester(eRequester := eRequester, bSourceLocked := FALSE, bFaulted := FALSE);
IF Advance <> E_RpcMethodResponse.ACCEPTED THEN RETURN; END_IF;
_SyncConfiguration();
IF _abortPending THEN
    Advance := E_RpcMethodResponse.REJECTED_INTERLOCKED;
    RETURN;
END_IF;
Advance := F_ValidateRequester(eRequester, bSourceLockedToProg, IsFaulted());
IF Advance <> E_RpcMethodResponse.ACCEPTED THEN RETURN; END_IF;
IF currentState = E_TwoPosActuator_State.Retracting THEN
    Advance := E_RpcMethodResponse.REJECTED_WRONG_STATE;
    RETURN;
END_IF;

IF (currentState = E_TwoPosActuator_State.Advanced AND NOT _inhibited) OR currentState = E_TwoPosActuator_State.Advancing THEN
    Advance := E_RpcMethodResponse.REJECTED_ALREADY_AT_TARGET;
    RETURN;
END_IF;

IF NOT advancePermissives.sts.bOK THEN
    Advance := E_RpcMethodResponse.REJECTED_PERMISSIVE_NOT_MET;
    RETURN;
END_IF;

_inhibited := FALSE;
currentState := E_TwoPosActuator_State.Advancing;
advanceTimer(IN := FALSE);
_AcceptCommand(eRequester := eRequester);
Advance := E_RpcMethodResponse.ACCEPTED;
END_METHOD

METHOD PUBLIC Retract : E_RpcMethodResponse
VAR_INPUT
    eRequester : E_Requester := E_Requester.PROG;
END_VAR
// Reject invalid identity before any command-specific mutation.
Retract := F_ValidateRequester(eRequester := eRequester, bSourceLocked := FALSE, bFaulted := FALSE);
IF Retract <> E_RpcMethodResponse.ACCEPTED THEN RETURN; END_IF;
_SyncConfiguration();
IF _abortPending THEN
    Retract := E_RpcMethodResponse.REJECTED_INTERLOCKED;
    RETURN;
END_IF;
Retract := F_ValidateRequester(eRequester, bSourceLockedToProg, IsFaulted());
IF Retract <> E_RpcMethodResponse.ACCEPTED THEN RETURN; END_IF;
IF currentState = E_TwoPosActuator_State.Advancing THEN
    Retract := E_RpcMethodResponse.REJECTED_WRONG_STATE;
    RETURN;
END_IF;

IF (currentState = E_TwoPosActuator_State.Retracted AND NOT _inhibited) OR currentState = E_TwoPosActuator_State.Retracting THEN
    Retract := E_RpcMethodResponse.REJECTED_ALREADY_AT_TARGET;
    RETURN;
END_IF;

IF NOT retractPermissives.sts.bOK THEN
    Retract := E_RpcMethodResponse.REJECTED_PERMISSIVE_NOT_MET;
    RETURN;
END_IF;

_inhibited := FALSE;
currentState := E_TwoPosActuator_State.Retracting;
retractTimer(IN := FALSE);
_AcceptCommand(eRequester := eRequester);
Retract := E_RpcMethodResponse.ACCEPTED;
END_METHOD

// Safety command — always accepted (bypasses source lock and fault check).
// De-energizes both valves and returns to Undefined for re-evaluation.
METHOD PUBLIC Abort : E_RpcMethodResponse
VAR_INPUT
    eRequester : E_Requester := E_Requester.PROG;
END_VAR
// Reject invalid identity before any command-specific mutation.
Abort := F_ValidateRequester(eRequester := eRequester, bSourceLocked := FALSE, bFaulted := FALSE);
IF Abort <> E_RpcMethodResponse.ACCEPTED THEN RETURN; END_IF;
_SyncConfiguration();
_operatorMailbox.CancelNormal();
outAdvance := FALSE;
outRetract := FALSE;
advanceTimer(IN := FALSE);
retractTimer(IN := FALSE);
_abortPending := TRUE;
_inhibited := TRUE;
outAdvance := FALSE; outRetract := FALSE;
currentState := E_TwoPosActuator_State.Undefined;
_AcceptCommand(eRequester := eRequester);
Abort := E_RpcMethodResponse.ACCEPTED;
END_METHOD

// Safety invariant: Reset is always accepted from any requester regardless
// of source lock or current state. Clears the active fault via the base and
// returns the device to Undefined so the body can re-evaluate feedback.
METHOD PUBLIC Reset : E_RpcMethodResponse
VAR_INPUT
    eRequester : E_Requester := E_Requester.PROG;
END_VAR
// Reject invalid identity before any command-specific mutation.
Reset := F_ValidateRequester(eRequester := eRequester, bSourceLocked := FALSE, bFaulted := FALSE);
IF Reset <> E_RpcMethodResponse.ACCEPTED THEN RETURN; END_IF;
_SyncConfiguration();
_operatorMailbox.CancelNormal();
SUPER^.Reset(eRequester := eRequester);

_abortPending := TRUE;
_inhibited := TRUE;
outAdvance := FALSE; outRetract := FALSE;
currentState := E_TwoPosActuator_State.Undefined;
outAdvance := FALSE;
outRetract := FALSE;
advanceTimer(IN := FALSE);
retractTimer(IN := FALSE);
Reset := E_RpcMethodResponse.ACCEPTED;
END_METHOD

// Translates this device's fault enum to human-readable text.
// Called by FB_DeviceBase to populate sts.header.faultString / lastFaultString.
METHOD PROTECTED ResolveFaultString : STRING(79)
VAR_INPUT
    code : DINT;
END_VAR
CASE code OF
    E_TwoPosActuator_Fault.BadConfig: ResolveFaultString := 'Actuator timeouts must be positive';
    E_TwoPosActuator_Fault.None:                ResolveFaultString := 'No Fault';
    E_TwoPosActuator_Fault.AdvanceTimeout:      ResolveFaultString := 'Advance Timeout';
    E_TwoPosActuator_Fault.RetractTimeout:      ResolveFaultString := 'Retract Timeout';
    E_TwoPosActuator_Fault.BothFeedbackOn:      ResolveFaultString := 'Both Feedbacks Active';
    E_TwoPosActuator_Fault.UndefinedState:      ResolveFaultString := 'Position Undefined';
    E_TwoPosActuator_Fault.PermissivesNotOK:    ResolveFaultString := 'Permissives Not OK';
    E_TwoPosActuator_Fault.ConflictingCommands: ResolveFaultString := 'Conflicting Commands';
    E_TwoPosActuator_Fault.NoFeedback:          ResolveFaultString := 'No Position Feedback';
ELSE
    ResolveFaultString := 'Unknown Fault';
END_CASE;
END_METHOD

METHOD PRIVATE _StateToString : STRING(31)
VAR_INPUT
    state : E_TwoPosActuator_State;
END_VAR
CASE state OF
    E_TwoPosActuator_State.Undefined:  _StateToString := 'Undefined';
    E_TwoPosActuator_State.Retracted:  _StateToString := 'Retracted';
    E_TwoPosActuator_State.Advancing:  _StateToString := 'Advancing';
    E_TwoPosActuator_State.Advanced:   _StateToString := 'Advanced';
    E_TwoPosActuator_State.Retracting: _StateToString := 'Retracting';
    E_TwoPosActuator_State.Fault:      _StateToString := 'Fault';
ELSE
    _StateToString := 'Unknown';
END_CASE;
END_METHOD

{attribute 'TcRpcEnable' := '1'}
METHOD PUBLIC OperatorAdvance : E_RpcMethodResponse

VAR_INPUT requestId : ULINT; END_VAR
OperatorAdvance := _operatorMailbox.Submit(requestId := requestId, command := E_OperatorCommand.Advance, value := 0.0);
END_METHOD

{attribute 'TcRpcEnable' := '1'}
METHOD PUBLIC OperatorRetract : E_RpcMethodResponse

VAR_INPUT requestId : ULINT; END_VAR
OperatorRetract := _operatorMailbox.Submit(requestId := requestId, command := E_OperatorCommand.Retract, value := 0.0);
END_METHOD

{attribute 'TcRpcEnable' := '1'}
METHOD PUBLIC OperatorAbort : E_RpcMethodResponse

VAR_INPUT requestId : ULINT; END_VAR
OperatorAbort := _operatorMailbox.Submit(requestId := requestId, command := E_OperatorCommand.Abort, value := 0.0);
END_METHOD

{attribute 'TcRpcEnable' := '1'}
METHOD PUBLIC OperatorReset : E_RpcMethodResponse

VAR_INPUT requestId : ULINT; END_VAR
OperatorReset := _operatorMailbox.Submit(requestId := requestId, command := E_OperatorCommand.Reset, value := 0.0);
END_METHOD

METHOD PUBLIC MapAdvanceCondition
VAR_INPUT
    bitIndex : UDINT;
    bGood : BOOL;
END_VAR
advancePermissives.MapInput(bitIndex := bitIndex, inputValue := bGood);
END_METHOD

METHOD PUBLIC MapRetractCondition
VAR_INPUT
    bitIndex : UDINT;
    bGood : BOOL;
END_VAR
retractPermissives.MapInput(bitIndex := bitIndex, inputValue := bGood);
END_METHOD

METHOD PROTECTED _DispatchOperatorCommand : E_RpcMethodResponse
VAR_INPUT command : E_OperatorCommand; value : REAL; END_VAR
CASE command OF
E_OperatorCommand.Advance: _DispatchOperatorCommand := THIS^.Advance(eRequester := E_Requester.OPERATOR);
E_OperatorCommand.Retract: _DispatchOperatorCommand := THIS^.Retract(eRequester := E_Requester.OPERATOR);
E_OperatorCommand.Abort: _DispatchOperatorCommand := THIS^.Abort(eRequester := E_Requester.OPERATOR);
ELSE _DispatchOperatorCommand := SUPER^._DispatchOperatorCommand(command := command, value := value);
END_CASE;
END_METHOD

METHOD PRIVATE _SyncConfiguration
// Configuration is owned by the same cyclic task as this device.
// The first observation establishes a baseline and preserves first-scan commands.
IF NOT _configurationKnown THEN
    _lastConfiguration := cfg;
    _configurationKnown := TRUE;
    RETURN;
END_IF;
IF cfg.advTimeoutS <> _lastConfiguration.advTimeoutS OR
   cfg.retTimeoutS <> _lastConfiguration.retTimeoutS OR
   cfg.holdAtAdvanced <> _lastConfiguration.holdAtAdvanced OR
   cfg.holdAtRetracted <> _lastConfiguration.holdAtRetracted THEN
    // Discard old operating intent before interpreting it under a new configuration.
    _operatorMailbox.CancelNormal();
    _inhibited := TRUE;
    advanceTimer(IN := FALSE);
    retractTimer(IN := FALSE);
    outAdvance := FALSE;
    outRetract := FALSE;
    // Re-observe position without retaining travel or hold intent; faults remain latched.
    currentState := E_TwoPosActuator_State.Undefined;
END_IF;
_lastConfiguration := cfg;
END_METHOD

END_FUNCTION_BLOCK

// ---- POUs/Base/FB_DeviceBase.TcPOU
// Abstract base for TcForge device-like function blocks. Provides:
//   - built-in fault book-keeping (current + last + persistent ring buffer)
//   - the source-lock flag (bSourceLockedToProg)
//   - safety-command primitives (Reset) that are always accepted
//   - diagnostics methods (IsFaulted / GetFaultCode / GetFaultString)
//   - protected helpers for children to populate ST_DeviceHeader_Sts
//
// Children:
//   - EXTEND this FB and declare their own sts containing ST_DeviceHeader_Sts
//     as the first member named `header`
//   - override ResolveFaultString(code) to map their device-specific fault
//     enum to human-readable text
//   - call _Raise(code, source, reason) to register a fault (idempotent on
//     `code`); _ClearFault() to clear without losing history
//   - call _AcceptCommand(eRequester) at the end of every accepted method
//   - call _UpdateHeader(sts.header, ...) once per cycle from the body
//
// Fault semantics:
//   - _Raise is idempotent on `code`. Repeated calls with the same non-zero
//     code push only one ring entry per episode; a different code replaces
//     the current fault and pushes a new entry (so a progression like
//     Timeout -> OddStep is preserved).
//   - _ClearFault wipes the active fault only. last* fields and the ring
//     survive so HMIs can still show what happened.
//   - The last-fault fields and ring buffer are PERSISTENT so that a process
//     restart does not silently lose the most recent fault context.
FUNCTION_BLOCK ABSTRACT FB_DeviceBase
VAR CONSTANT
    FAULT_RING_SIZE : UDINT := 8;
END_VAR

VAR
    {attribute 'OPC.UA.DA' := '0'}
    _operatorMailbox : FB_OperatorMailbox;
    {attribute 'OPC.UA.DA' := '0'}
    bSourceLockedToProg : BOOL;
    {attribute 'OPC.UA.DA' := '0'}
    _lastRequester : E_Requester;
    {attribute 'OPC.UA.DA' := '0'}
    _tsLastCommand : LTIME;

    // Active fault (not persistent; Reset on restart so recovery logic re-runs).
    {attribute 'OPC.UA.DA' := '0'}
    _faultCode   : DINT;
    {attribute 'OPC.UA.DA' := '0'}
    _faultTs     : LTIME;
    {attribute 'OPC.UA.DA' := '0'}
    _faultSource : STRING(31);
    {attribute 'OPC.UA.DA' := '0'}
    _faultReason : STRING(79);
END_VAR

VAR PERSISTENT
    // Most recent fault — survives Reset (and PLC restart) so HMIs can always
    // show "last fault info".
    _lastFaultCode      : DINT;
    _lastFaultTs        : LTIME;
    _lastFaultRequester : E_Requester;
    _lastFaultSource    : STRING(31);
    _lastFaultReason    : STRING(79);

    // Short ring-buffer history.
    _faultRing     : ARRAY[0..7] OF ST_FaultEntry;
    _faultRingHead : UDINT;
END_VAR

// Abstract base — children implement their own cyclic logic.

// Base Reset clears diagnostics from any requester, regardless
// of source lock or current fault state. Clears the active fault; history is
// preserved in the ring buffer. Children may override to add device-specific
// recovery validation and cleanup. Successful overrides call SUPER^.Reset;
// the state machine rejects Reset until STOPPED and running conditions are good.
METHOD PUBLIC Reset : E_RpcMethodResponse
VAR_INPUT
    eRequester : E_Requester := E_Requester.PROG;
END_VAR
// Reject invalid identity before any command-specific mutation.
Reset := F_ValidateRequester(eRequester := eRequester, bSourceLocked := FALSE, bFaulted := FALSE);
IF Reset <> E_RpcMethodResponse.ACCEPTED THEN RETURN; END_IF;
_operatorMailbox.CancelNormal();
_ClearFault();
_AcceptCommand(eRequester := eRequester);
Reset := E_RpcMethodResponse.ACCEPTED;
END_METHOD

METHOD PUBLIC LockSource : E_RpcMethodResponse
VAR_INPUT
    bLock : BOOL;
END_VAR
bSourceLockedToProg := bLock;
LockSource := E_RpcMethodResponse.ACCEPTED;
END_METHOD

METHOD PUBLIC IsFaulted : BOOL
IsFaulted := _faultCode <> 0;
END_METHOD

METHOD PUBLIC GetFaultCode : DINT
GetFaultCode := _faultCode;
END_METHOD

METHOD PUBLIC GetFaultString : STRING(79)
// Virtual dispatch: child's ResolveFaultString() maps the current code.
GetFaultString := THIS^.ResolveFaultString(code := _faultCode);
END_METHOD

// Children override to translate their fault-enum value into human-readable
// text. Default returns empty so devices without a fault model still compile.
METHOD PROTECTED ResolveFaultString : STRING(79)
VAR_INPUT
    code : DINT;
END_VAR
ResolveFaultString := '';
END_METHOD

// Book-keeping called at the end of every accepted command method.
METHOD PROTECTED _AcceptCommand
VAR_INPUT
    eRequester : E_Requester;
END_VAR
_lastRequester := eRequester;
_tsLastCommand := F_Now();
END_METHOD

// Raise a fault with optional source (where it came from) and reason (free-form).
// Idempotent on `code`: a second call with the same non-zero code in the
// same episode is a no-op (returns FALSE) even if source/reason differ — so
// cyclic callers can spam this without flooding the ring. A different
// non-zero code replaces the current fault and pushes a new ring entry.
// The requester recorded with the fault is the most recent command requester
// (_lastRequester), which is what the operator / HMI has context for.
// Returns TRUE when a new ring entry was pushed this call.
METHOD PROTECTED _Raise : BOOL
VAR_INPUT
    code   : DINT;
    source : STRING(31);
    reason : STRING(79);
END_VAR
IF code = 0 THEN
    _Raise := FALSE;
    RETURN;
END_IF;

IF code = _faultCode THEN
    _Raise := FALSE;
    RETURN;
END_IF;

_faultCode   := code;
_faultTs     := F_Now();
_faultSource := source;
_faultReason := reason;

_lastFaultCode      := code;
_lastFaultTs        := _faultTs;
_lastFaultRequester := _lastRequester;
_lastFaultSource    := source;
_lastFaultReason    := reason;

_faultRingHead := _faultRingHead MOD FAULT_RING_SIZE;
_faultRing[_faultRingHead].code      := code;
_faultRing[_faultRingHead].ts        := _faultTs;
_faultRing[_faultRingHead].requester := _lastRequester;
_faultRing[_faultRingHead].source    := source;
_faultRing[_faultRingHead].reason    := reason;
_faultRingHead := (_faultRingHead + 1) MOD FAULT_RING_SIZE;

_Raise := TRUE;
END_METHOD

// Clear the currently-active fault. Preserves the ring buffer and the
// last-fault fields so HMIs can still show what happened.
METHOD PROTECTED _ClearFault
_faultCode   := 0;
_faultTs     := LTIME#0ns;
_faultSource := '';
_faultReason := '';
END_METHOD

// Refreshes the common header a child embeds as `header` in its sts struct.
// Call once per cycle from the child's cyclic body. Device-specific fields
// (advanced, value, etc.) stay in the child sts alongside `header`.
METHOD PROTECTED _UpdateHeader
VAR_IN_OUT
    header : ST_DeviceHeader_Sts;
END_VAR
VAR_INPUT
    stateString : STRING(31);
    busy     : BOOL;
END_VAR
header.stateString     := stateString;
header.busy         := busy;
header.faulted      := _faultCode <> 0;
header.ready        := NOT header.faulted AND NOT busy AND NOT bSourceLockedToProg;
header.sourceLocked := bSourceLockedToProg;
header.faultCode       := _faultCode;
header.faultString     := THIS^.ResolveFaultString(code := _faultCode);
header.faultSource     := _faultSource;
header.faultReason     := _faultReason;
header.lastFaultCode   := _lastFaultCode;
header.lastFaultString := THIS^.ResolveFaultString(code := _lastFaultCode);
header.lastFaultSource := _lastFaultSource;
header.lastFaultReason := _lastFaultReason;
header.lastRequester   := _lastRequester;
header.tsLastCommand   := _tsLastCommand;
header.tsLastFault     := _lastFaultTs;
END_METHOD

{attribute 'TcRpcEnable' := '1'}
METHOD PUBLIC OperatorReset : E_RpcMethodResponse

VAR_INPUT requestId : ULINT; END_VAR
OperatorReset := _operatorMailbox.Submit(requestId := requestId, command := E_OperatorCommand.Reset, value := 0.0);
END_METHOD

{attribute 'TcRpcEnable' := '1'}
METHOD PUBLIC OperatorCommandResult : E_RpcMethodResponse
VAR_INPUT requestId : ULINT; END_VAR
OperatorCommandResult := _operatorMailbox.GetResult(requestId := requestId);
END_METHOD

METHOD PROTECTED _ProcessOperatorCommands
VAR command : E_OperatorCommand; value : REAL; result : E_RpcMethodResponse; END_VAR
IF _operatorMailbox.BeginConsume(command => command, value => value) THEN
    result := THIS^._DispatchOperatorCommand(command := command, value := value);
    _operatorMailbox.EndConsume(result := result);
END_IF;
END_METHOD

METHOD PROTECTED _DispatchOperatorCommand : E_RpcMethodResponse
VAR_INPUT command : E_OperatorCommand; value : REAL; END_VAR
CASE command OF
E_OperatorCommand.Reset: _DispatchOperatorCommand := THIS^.Reset(eRequester := E_Requester.OPERATOR);
ELSE _DispatchOperatorCommand := E_RpcMethodResponse.REJECTED_INVALID_PARAMETER;
END_CASE;
END_METHOD

END_FUNCTION_BLOCK

